(* CODESYS project Git_Repo
   Author: SESA110233
   DefaultNamespace: CrankModuleExample
   Title: Template_GitHub_ESME22
   Version: 0.0.0.0

Project tree, tasks and I/O mapping:
  LMC_PacDrive : PacDrive LMC 300/400/402/600/802/902C, Schneider Electric, order no. LMC Pro and Pro2, version 1.76.4.3
    application Application
      libraries: PD_GlobalDiagnostics, 1.6.0.0 (Schneider Electric); PD_PacDriveLib, 1.10.3.0 (Schneider Electric); PD_Template, 1.8.0.0 (Schneider Electric); PD_AxisModule, 1.7.1.0 (Schneider Electric); CrankModule, 1.4.1.0 (Schneider Electric); ApplicationLogger, 1.1.7.0 (Schneider Electric); IecRtsServices, 1.0.5.0 (Schneider Electric)
      task TASK_SR_Diagnostics (cyclic, interval T#100ms, priority 31, watchdog T#100ms x 2) calls SR_Diagnostics
      task TASK_SR_Logging (cyclic, interval T#10ms, priority 13, watchdog T#10ms x 2) calls SR_Logging
      task TASK_SR_MainMachine (cyclic, interval T#10ms, priority 8, watchdog t#10ms x 10) calls SR_HWCopyIO, SR_MainMachine
      task TASK_SR_VisControl (cyclic, interval T#50ms, priority 14, watchdog T#50ms x 2) calls SR_VisControl
      function CheckBounds [ST]
      function CheckDivDInt [ST]
      function CheckDivLInt [ST]
      function CheckDivLReal [ST]
      function CheckDivReal [ST]
      function CheckLRangeSigned [ST]
      function CheckLRangeUnsigned [ST]
      function CheckPointer [ST]
      function CheckRangeSigned [ST]
      function CheckRangeUnsigned [ST]
      CrankModuleExample/
        EquipmentModules/
          program SR_AlphaModule [SFC]: ExceptionControl_Action, Init_CmdTables, Init_Exceptions, Init_Master, Init_Reactions, Init_SubModules, InitModule_Action, Input_Action, Logger_Action, ModuleFaults, Output_Active, Start_Action, SubModules_Action, UpdateStructs
          program SR_BravoModule [SFC]: ExceptionControl_Action, Init_CmdTables, Init_Exceptions, Init_Reactions, Init_Slave1, Init_Slave2, Init_SubModules, InitModule_Action, Input_Action, Logger_Action, ModuleFaults, Output_Active, Start_Action, SubModules_Action, UpdateStructs
          program SR_CharlyModule [SFC]: ExceptionControl_Action, Init_CmdTables, Init_CrankModule, Init_Exceptions, Init_Nocke1, Init_Reactions, Init_Slave3, Init_Slave4, Init_SubModules, InitModule_Action, Input_Action, Logger_Action, Logic_Action, ModuleFaults, Output_Active, Start_Action, SubModules_Action, UpdateStructs
          program SR_NodeWithoutMotionModule [SFC]: ExceptionControl_Action, Init_CmdTables, Init_Exceptions, Init_Reactions, Init_SubModules, InitModule_Action, Input_Action, Logger_Action, ModuleFaults, Output_Active, Start_Action, SubModules_Action, UpdateStructs
        Examples/
          ExampleCmds/
            data type ET_Cmd
          ExampleModulesExtItf/
            function block FB_AxisModuleExtItf [ST]
            function block FB_ExampleLeafModuleExtItf [ST]
            function block FB_ExampleNodeFbModuleExtItf [ST]
            program SR_CharlyModuleExtItf [ST]
          ExampleNodeAsFB/
            function block FB_ExampleNodeFbModule [SFC]: ExceptionControl_Action, Init_CmdTables, Init_Exceptions, Init_Reactions, Init_Slave1, Init_Slave2, Init_SubModules, InitModule_Action, Input_Action, Logger_Action, ModuleFaults, Output_Active, Start_Action, SubModules_Action, UpdateStructs
            data type ST_ExampleNodeAsFbInterface
        GlobalVariables/
          global variables Diagnostics
          global variables ExceptionHandling
          global variables HardwareInOuts
          global variables InputVariablesEpas
          global variables InputVariablesExt
          global variables IntelligentLineShaft
          global variables Logging
          global variables RestoreAxisPosition
        ProjectDiagnostics/
          data type ET_DiagExt
          data type ET_DiagExtUser
          function FC_EtDiagExtToString [ST]
          function FC_EtDiagExtUserToString [ST]
        TaskCalls/
          program SR_Diagnostics [FBD]: SetDiagnosticsWarning
          program SR_HWCopyIO [FBD]
          program SR_Logging [FBD]
          program SR_MainMachine [SFC]: _aStart_active, AutoStep_Action, AutoStep_Entry, AutoStop_Action, AutoStop_Entry, BrakeReleaseStep_Action, BrakeReleaseStep_Entry, ExceptionControl_Action, Init_Alpha, Init_Bravo, Init_Charly, Init_CmdTables, Init_Exceptions, Init_NodeWithoutMotion, Init_Reactions, Init_SubModules, InitModule_Action, Input_Action, JogMachineStep_Action, JogMachineStep_Entry, Logger_Action, Logic_active, MainSystemFaults, MainUserFaults, ManualStep_Action, ManualStep_Entry, ModeSelect_Action, Output_Action, PrepStep_Action, PrepStep_Entry, PrepStop_Action, PrepStop_Entry, StopBrake_Action, StopBrake_Entry, StopJog_Action, StopJog_Entry, StopMan_Action, StopMan_Entry, SubModules_Action, UpdateStructs
          program SR_VisControl [ST]: CallTestErrors, CrankModuleVis, CurrentModuleCmdTable, DetectOpModeChange, ExceptionVis, InitTestExceptions, LoggerVis, MainPageCmdTable, ModuleNavigationIn, ModuleNavigationOut, ModuleReaction, ModuleVisController, OpModeControl, SearchCurrentModule, SetCurrentModule
        Tools/
          function FC_IsDriveVirtual [ST]
          function FC_SetDeadTimeCompensation [ST]
        Visualization/
          CrankModule/
            visualisation VIS_CrankModule
          visualisation VIS_Main
      function block FB_ExampleTableDiagSource [ST]: CancelWriting, ExceptionDuringWriting, SetDiagOutputs
      function block FB_ExampleTreeDiagSource [ST]: CancelWriting, ExceptionDuringWriting, SetDiagOutputs
      data type ET_DiagExtExampleLeafModule
      data type ET_ExampleLeafModuleCmd
      data type ET_ExampleLeafModuleState
      data type ET_ExceptionSource
      data type ET_ModuleType
      function block FB_ExampleLeafModule [SFC]: Auto_Action, Auto_Entry, CancelException, CheckCmd, CmdControl_Action, DiagQuit, DisableAllJobs, ExceptionHandler_Action, Homing_Action, Homing_Entry, InactiveCmdExecution, Init_Action, InitHoming_Action, InitHoming_Entry, Input_Action, Logger_Action, NoOp_Entry, Output_Active, RefuseCommand, ReportException, SetInterfaces, SetOutputs, SignalSuccessfulExecution, SignalUnSuccessfulExecution
      function block FB_ExampleLeafModuleController [ST]
      function block FB_ExampleLeafModuleVisController [ST]
      function FC_EtDiagExtExampleLeafModuleToString [ST]
      function FC_EtExampleLeafModuleCmdToString [ST]
      function FC_EtExampleLeafModuleStateToString [ST]
      function FC_UpdateExampleLeafModuleAddInterfaceStruct [ST]
      data type ST_ExampleLeafModuleInterface
      visualisation FR_ButtonAssignId
      visualisation FR_ExampleLeafModule
      visualisation FR_ExampleLeafModuleSelect
      visualisation VIS_ExampleLeafModule
      visualisation FR_ControlModuleTypes
      visualisation FR_NavigationButtons
      visualisation FR_OtherModuleTypes
      visualisation VIS_AxisModule
      visualisation VIS_ControlModule
      visualisation VIS_ExceptionDetails
      visualisation VIS_ExceptionList
      visualisation VIS_LogDataList
      visualisation VIS_LogDataListExt
      visualisation VIS_ModuleDetails
      visualisation VIS_ModuleExceptions
      visualisation VIS_Modules
      visualisation VIS_VisNavigation
    Device Addressing
    Message Logger
    AI_0 : Analog Input, Schneider Electric, version 1.76.4.3
    AI_1 : Analog Input, Schneider Electric, version 1.76.4.3
    AQ_0 : Analog Output, Schneider Electric, version 1.76.4.3
    AQ_1 : Analog Output, Schneider Electric, version 1.76.4.3
    DIG_DigitalIn : Digital Inputs, Schneider Electric, version 1.76.4.3
      DI_0 : Input, Schneider Electric, version 1.76.4.3
      DI_10 : Input, Schneider Electric, version 1.76.4.3
      DI_11 : Input, Schneider Electric, version 1.76.4.3
      DI_12 : Input, Schneider Electric, version 1.76.4.3
      DI_13 : Input, Schneider Electric, version 1.76.4.3
      DI_14 : Input, Schneider Electric, version 1.76.4.3
      DI_15 : Input, Schneider Electric, version 1.76.4.3
      DI_16 : Input, Schneider Electric, version 1.76.4.3
      DI_17 : Input, Schneider Electric, version 1.76.4.3
      DI_18 : Input, Schneider Electric, version 1.76.4.3
      DI_19 : Input, Schneider Electric, version 1.76.4.3
      DI_1 : Input, Schneider Electric, version 1.76.4.3
      DI_2 : Input, Schneider Electric, version 1.76.4.3
      DI_3 : Input, Schneider Electric, version 1.76.4.3
      DI_4 : Input, Schneider Electric, version 1.76.4.3
      DI_5 : Input, Schneider Electric, version 1.76.4.3
      DI_6 : Input, Schneider Electric, version 1.76.4.3
      DI_7 : Input, Schneider Electric, version 1.76.4.3
      DI_8 : Input, Schneider Electric, version 1.76.4.3
      DI_9 : Input, Schneider Electric, version 1.76.4.3
      FI_0 : Fast Input, Schneider Electric, version 1.76.4.3
      FI_1 : Fast Input, Schneider Electric, version 1.76.4.3
      FI_2 : Fast Input, Schneider Electric, version 1.76.4.3
      FI_3 : Fast Input, Schneider Electric, version 1.76.4.3
    DQG_DigitalOut : Digital Outputs, Schneider Electric, version 1.76.4.3
        settings: OpenloadDiagMsk = 0
      DQ_0 : Output, Schneider Electric, version 1.76.4.3
      DQ_10 : Output, Schneider Electric, version 1.76.4.3
      DQ_11 : Output, Schneider Electric, version 1.76.4.3
      DQ_12 : Output, Schneider Electric, version 1.76.4.3
      DQ_13 : Output, Schneider Electric, version 1.76.4.3
      DQ_14 : Output, Schneider Electric, version 1.76.4.3
      DQ_15 : Output, Schneider Electric, version 1.76.4.3
      DQ_1 : Output, Schneider Electric, version 1.76.4.3
      DQ_2 : Output, Schneider Electric, version 1.76.4.3
      DQ_3 : Output, Schneider Electric, version 1.76.4.3
      DQ_4 : Output, Schneider Electric, version 1.76.4.3
      DQ_5 : Output, Schneider Electric, version 1.76.4.3
      DQ_6 : Output, Schneider Electric, version 1.76.4.3
      DQ_7 : Output, Schneider Electric, version 1.76.4.3
      DQ_8 : Output, Schneider Electric, version 1.76.4.3
      DQ_9 : Output, Schneider Electric, version 1.76.4.3
    LE_EncCrank : Log. Encoder, Schneider Electric, version 1.76.4.3
    LE_EncSlide : Log. Encoder, Schneider Electric, version 1.76.4.3
    LE_Master : Log. Encoder, Schneider Electric, version 1.76.4.3
    LE_Slave1 : Log. Encoder, Schneider Electric, version 1.76.4.3
    LE_Slave2 : Log. Encoder, Schneider Electric, version 1.76.4.3
    LE_Slave3 : Log. Encoder, Schneider Electric, version 1.76.4.3
    LE_Slave4 : Log. Encoder, Schneider Electric, version 1.76.4.3
    Sercos_Master : Sercos Master, Schneider Electric, version 1.76.4.3
      DRV_CrankDrive : Lexium LXM62 Drive, Schneider Electric, order no. LXM62DU60, LXM62DD15, LXM62DD27, LXM62DD45, LXM62DC13, version 1.76.4.3
      DRV_Master : Lexium LXM62 Drive, Schneider Electric, order no. LXM62DU60, LXM62DD15, LXM62DD27, LXM62DD45, LXM62DC13, version 1.76.4.3
      DRV_Slave1 : Lexium LXM62 Drive, Schneider Electric, order no. LXM62DU60, LXM62DD15, LXM62DD27, LXM62DD45, LXM62DC13, version 1.76.4.3
      DRV_Slave2 : Lexium LXM62 Drive, Schneider Electric, order no. LXM62DU60, LXM62DD15, LXM62DD27, LXM62DD45, LXM62DC13, version 1.76.4.3
      DRV_Slave3 : Lexium LXM62 Drive, Schneider Electric, order no. LXM62DU60, LXM62DD15, LXM62DD27, LXM62DD45, LXM62DC13, version 1.76.4.3
      DRV_Slave4 : Lexium LXM62 Drive, Schneider Electric, order no. LXM62DU60, LXM62DD15, LXM62DD27, LXM62DD45, LXM62DC13, version 1.76.4.3
      DRV_SlideDrive : Lexium LXM62 Drive, Schneider Electric, order no. LXM62DU60, LXM62DD15, LXM62DD27, LXM62DD45, LXM62DC13, version 1.76.4.3
      PSM_PowerSupply : Lexium LXM62 Power Supply, Schneider Electric, order no. LXM62PD84, LXM62PD20, version 1.76.4.3
    TPG_TPIn : Touch Probe Inputs, Schneider Electric, version 1.76.4.3
      TP_0 : Touch Probe Input, Schneider Electric, version 1.76.4.3
      TP_10 : Touch Probe Input, Schneider Electric, version 1.76.4.3
      TP_11 : Touch Probe Input, Schneider Electric, version 1.76.4.3
      TP_12 : Touch Probe Input, Schneider Electric, version 1.76.4.3
      TP_13 : Touch Probe Input, Schneider Electric, version 1.76.4.3
      TP_14 : Touch Probe Input, Schneider Electric, version 1.76.4.3
      TP_15 : Touch Probe Input, Schneider Electric, version 1.76.4.3
      TP_1 : Touch Probe Input, Schneider Electric, version 1.76.4.3
      TP_2 : Touch Probe Input, Schneider Electric, version 1.76.4.3
      TP_3 : Touch Probe Input, Schneider Electric, version 1.76.4.3
      TP_4 : Touch Probe Input, Schneider Electric, version 1.76.4.3
      TP_5 : Touch Probe Input, Schneider Electric, version 1.76.4.3
      TP_6 : Touch Probe Input, Schneider Electric, version 1.76.4.3
      TP_7 : Touch Probe Input, Schneider Electric, version 1.76.4.3
      TP_8 : Touch Probe Input, Schneider Electric, version 1.76.4.3
      TP_9 : Touch Probe Input, Schneider Electric, version 1.76.4.3
  00000000-0000-0000-0000-000000000000|M:\lib-jenkins-config\externalfiles\Disclaimer of Warranty.pdf
  Disclaimer of Warranty
  text list GlobalTextList
  function GetBooleanProperty [ST]
  function GetTextProperty2 [ST]
  function GetTextProperty [ST]
  function GetTitle [ST]
*)

// LMC_PacDrive/Application/CrankModuleExample/ProjectDiagnostics/ET_DiagExt
{attribute 'qualified_only'}
TYPE ET_DiagExt :
(
	(* Minimum value +0 *)
	Ok								:= 0,
	Disabled						:= 1,
	WaitUntilControllerFinishedBoot	:= 2,
	Initializing					:= 3,
	DeactivatingSubModules			:= 4,
	ExecuteStep						:= 5,
	WaitAtNegativeStep				:= 6,
	WaitCmdsDone					:= 7,
	WaitForCmd						:= 8,
	SubModuleInException			:= 9,
	ModuleControllerException		:= 10,
	UnknownStateModuleController	:= 11,
	
	SystemFatalException			:= 12,
	SystemException					:= 13,
	SystemWarning					:= 14,
	MainSystemEmergencyStop			:= 15,
	InvalidPointer					:= 16,	
	UpdateStructsException			:= 17,
	InitReactionsException			:= 18,
	InitSubModulesException			:= 19,
	DriveInvalid					:= 20,
	UnknownDiagExt					:= 21,
	
	Exception1FromVis				:= 22,
	Exception2FromVis				:= 23,
	Exception3FromVis				:= 24,
	Exception4FromVis				:= 25,
	Exception5FromVis				:= 26,
	
	DiagnosticsWarning					:= 27,
	WaitUntilDiagnosticsManagerReady	:= 28,
	WaitUntilDisabled					:= 29,
	WaitUntilDiagSourceRegistered		:= 30,
	WaitForCommunication				:= 31,
	DataSuccessfullyWritten				:= 32,
	WritingToFile						:= 33,
	FileIdInvalid						:= 34,
	CmdUnknown							:= 35,	
	UnexpectedFeedback					:= 36,
	UnknownDiagExtUser					:= 37
)UDINT;
END_TYPE

// LMC_PacDrive/Application/CrankModuleExample/ProjectDiagnostics/ET_DiagExtUser
{attribute 'qualified_only'}
TYPE ET_DiagExtUser :
(
(* Minimum value +0 *)
	Exception1FromEquipmentModule		:= 0,
	Exception2FromEquipmentModule		:= 1,
	
	Exception1FromMain					:= 2,
	Exception2FromMain					:= 3,
	Exception3FromMain					:= 4,
	Exception4FromMain					:= 5,
	Exception5FromMain					:= 6
)UDINT;
END_TYPE

// LMC_PacDrive/Application/CrankModuleExample/Examples/ExampleCmds/ET_Cmd
{attribute 'qualified_only'}
TYPE ET_Cmd :
(	NoCmd				:= 0,

	(* TPL.Gc_udiUserCmdOffset : UDINT := 25000; // >= 25000: user defined Commands *)
	DriveEnableOn		:= 25999,
	DriveEnableOff		:= 25998,
	Init				:= 25997,
	Prepare				:= 25996,
	Production			:= 25995,
	Auto				:= 25994,
	BrakeRelease		:= 25993,
	Abort				:= 25992,
	Standby				:= 25991,
	Manual				:= 25990,
	Jogging				:= 25989,
	Hold				:= 25988,
	Stop				:= 25987,
	Start				:= 25986,
	HoldJM				:= 25985
);
END_TYPE

// LMC_PacDrive/Application/ET_DiagExtExampleLeafModule
{attribute 'qualified_only'}
TYPE ET_DiagExtExampleLeafModule :
(
(* Minimum value +0 *)
	Ok										:= 0,
	Disabled								:= 1,
	Initializing							:= 2,
	NoOp									:= 3,
	HomingWaitForStart						:= 4,
	HomingExecuting							:= 5,
	HomingDone								:= 6,
	AutoWaitForStart						:= 7,
	AutoRunning								:= 8,
	Working									:= 9,

	UnknownDiagExtExampleLeafModule			:= 10,
	SubModuleAddInterfacesInvalidPointer	:= 11,
	SubModuleConstantRange					:= 12,
	MissingExtInit							:= 13,
	ReactionOffsetRange						:= 14,
	DriveInvalid							:= 15,
	
	CmdUnknown								:= 16,
	CmdImpossibleOverwrite					:= 17,
	CmdImpossibleState						:= 18,
	CmdImpossibleReaction					:= 19,
	
	AsyncStop								:= 20,
	SyncStopEL								:= 21,
	SyncStopEH								:= 22,
	StopEndOfCycle							:= 23,
	
	DriveFatalException						:= 24,
	DriveException							:= 25,
	DriveWarning							:= 26,
	
	UnknownState							:= 27,
	UnknownCmd								:= 28,
	RandomException							:= 29,
	
	CurrentStandardItfInvalidPointer		:= 30,
	CurrentAddItfInvalidPointer				:= 31
)UDINT;
END_TYPE

// LMC_PacDrive/Application/ET_ExampleLeafModuleCmd
{attribute 'qualified_only'}
TYPE ET_ExampleLeafModuleCmd :
(
	(* TPL.Gc_udiUserCmdOffset : UDINT := 25000; // >= 25000: user defined Commands *)
	Homing				:= 30000,
	Auto				:= 30001,
	Start				:= 30002,
	Stop				:= 30003,
	Hold				:= 30004
	
)DINT; //UDINT;
END_TYPE

// LMC_PacDrive/Application/ET_ExampleLeafModuleState
{attribute 'qualified_only'}
TYPE ET_ExampleLeafModuleState :
(
	NoOp				:= 0,
	Disabled			:= 1,
	Initializing		:= 2,
	HomingWaitForStart	:= 3,
	HomingExecuting		:= 4,
	HomingDone			:= 5,
	AutoWaitForStart	:= 6,
	AutoRunning			:= 7
)UDINT;
END_TYPE

// LMC_PacDrive/Application/ET_ExceptionSource
{attribute 'qualified_only'}
TYPE ET_ExceptionSource :
(
	(* 0 - 9999 = reserved area *)
	
	(* Sources > 9999 = free Area *)
	ExampleLeafModule	:= 15000
)UDINT;
END_TYPE

// LMC_PacDrive/Application/ET_ModuleType
{attribute 'qualified_only'}
TYPE ET_ModuleType :
(
	(* 0 - 9999 = reserved area *)
	(* IDs >9999 = free Area *)
	ExampleLeafModule := 15000 (* Definition of the dwModuleType for the module *)
)UDINT;
END_TYPE

// LMC_PacDrive/Application/ST_ExampleLeafModuleInterface
TYPE ST_ExampleLeafModuleInterface :
STRUCT
	i_ifDrive						: SystemConfigurationItf.IF_Drive;
	i_lrPosMin						: LREAL;
	i_lrPosMax						: LREAL;
	i_xInitHoming					: BOOL;
	i_xEnableRandomExceptionTrigger	: BOOL;
	
	q_xValue						: BOOL := FALSE;
	q_etState						: ET_ExampleLeafModuleState := ET_ExampleLeafModuleState.Disabled;
END_STRUCT
END_TYPE

// LMC_PacDrive/Application/CrankModuleExample/Examples/ExampleNodeAsFB/ST_ExampleNodeAsFbInterface
TYPE ST_ExampleNodeAsFbInterface :
STRUCT
	i_ifSlave1				: SystemConfigurationItf.IF_Drive;
	i_lencEncoder1			: SystemConfiguration.L_ENC;
	i_ifHomingTouchProbe1	: SystemConfigurationItf.IF_TouchProbe;
	i_pstRestorePosRetain1	: POINTER TO PDL.ST_AxisRestorePosition;
	
	i_ifSlave2				: SystemConfigurationItf.IF_Drive;
	i_lencEncoder2			: SystemConfiguration.L_ENC;
	i_ifHomingTouchProbe2	: SystemConfigurationItf.IF_TouchProbe;
	i_pstRestorePosRetain2	: POINTER TO PDL.ST_AxisRestorePosition;
END_STRUCT
END_TYPE

// LMC_PacDrive/Application/CrankModuleExample/GlobalVariables/Diagnostics
VAR_GLOBAL
	G_stDiagnosticsToApplicationMarkerarea AT %MB0 : TPL.ST_DiagnosticsToApplicationMarkerArea;
END_VAR

// LMC_PacDrive/Application/CrankModuleExample/GlobalVariables/ExceptionHandling
VAR_GLOBAL
	G_stExceptionList		: TPL.ST_ExceptionList;
END_VAR

// LMC_PacDrive/Application/CrankModuleExample/GlobalVariables/HardwareInOuts
VAR_GLOBAL
	G_xMainsContactorOut 		(*-AT %QX0.0-*)	: BOOL;

	G_xEmergencyIn  			(*-AT %IX0.0-*)	: BOOL;
	G_xMainsContactorIn 		(*-AT %IX0.1-*)	: BOOL;
END_VAR

// LMC_PacDrive/Application/CrankModuleExample/GlobalVariables/InputVariablesEpas
VAR_GLOBAL
	G_xStartEpas				: BOOL;
	G_xStopEpas					: BOOL;
	G_xPrepareEpas				: BOOL;
	G_xAutoEpas					: BOOL;
	G_xHoldEpas					: BOOL;
	G_xAbortEpas				: BOOL;
	G_xProductsOkEpas			: BOOL;
	G_xPowerOnEpas				: BOOL;
	G_xPowerOffEpas				: BOOL;
	G_xManualEpas				: BOOL;
	G_xJogMachineEpas			: BOOL;
	G_xDiagQuitEpas				: BOOL;
	G_xEmergencyEpas			: BOOL := TRUE;
	G_xJogForwEpas				: BOOL;
	G_xJogBackEpas				: BOOL;
	G_xBrakeReleaseEpas			: BOOL;
	
	G_udiManualModuleSelect		: UDINT;

	G_xDoEnableVis				: BOOL;
	
	G_xDoEnableCrankVis			: BOOL; // created for Crank execution.

	G_xDoPrepare 				: BOOL;
	G_xDoAuto	 				: BOOL;
	G_xDoManual 				: BOOL;
	G_xDoJogMachine 			: BOOL;
	G_xDoBrakeRelease			: BOOL;

	G_xPrepareActive 			: BOOL;
	G_xAutoActive	 			: BOOL;
	G_xManualActive 			: BOOL;
	G_xJogMachineActive 		: BOOL;
	G_xBrakeReleaseActive		: BOOL;
END_VAR

// LMC_PacDrive/Application/CrankModuleExample/GlobalVariables/InputVariablesExt
VAR_GLOBAL
	G_xStartExt			: BOOL;
	G_xStopExt			: BOOL;
	G_xPrepareExt		: BOOL;
	G_xAutoExt			: BOOL;
	G_xHoldExt			: BOOL;
	G_xAbortExt			: BOOL;
	G_xProductsOkExt	: BOOL;
	G_xPowerOnExt		: BOOL;
	G_xPowerOffExt		: BOOL;
	G_xManualExt		: BOOL;
	G_xJogMachineExt	: BOOL;
	G_xDiagQuitExt		: BOOL;
	G_xJogForwExt		: BOOL;
	G_xJogBackExt		: BOOL;
	G_xBrakeReleaseExt	: BOOL;
END_VAR

// LMC_PacDrive/Application/CrankModuleExample/GlobalVariables/IntelligentLineShaft
VAR_GLOBAL
	G_stIlsData : PDL.ST_IlsData;
END_VAR

// LMC_PacDrive/Application/CrankModuleExample/GlobalVariables/Logging
VAR_GLOBAL
	G_stLogDataList			: TPL.ST_LogDataList;			(* Global log data list *)
	G_stLogDataListAscii	: TPL.ST_LogDataListAscii;		(* Temp.list for save in XML format *)
	G_stLoggerInterface		: TPL.ST_LoggerInterface;		(* Interface between logger and main machine *)
END_VAR

// LMC_PacDrive/Application/CrankModuleExample/GlobalVariables/RestoreAxisPosition
VAR_GLOBAL PERSISTENT RETAIN
	Grp_stRestorePositionAxis1		: PDL.ST_AxisRestorePosition;
	Grp_stRestorePositionAxis2		: PDL.ST_AxisRestorePosition;
	Grp_stRestorePositionAxis3		: PDL.ST_AxisRestorePosition;
	Grp_stRestorePositionAxis4		: PDL.ST_AxisRestorePosition;
	Grp_stRestorePositionAxis5		: PDL.ST_AxisRestorePosition;
	Grp_stRestorePositionAxis6		: PDL.ST_AxisRestorePosition;
	Grp_stRestorePositionAxis7		: PDL.ST_AxisRestorePosition;
	Grp_stRestorePositionAxis8		: PDL.ST_AxisRestorePosition;
	Grp_stRestorePositionAxisCrank	: PDL.ST_AxisRestorePosition;
END_VAR

// LMC_PacDrive/Application/CrankModuleExample/TaskCalls/SR_Diagnostics
PROGRAM SR_Diagnostics
VAR
	fbDiagnosticsManager : TPL.FB_DiagnosticsManager;
	stComStructure 		 : TPL.ST_DiagnosticsManagerToDiagSource;
	
	stWarning 		: TPL.ST_Exception;
	etLastDiagExt	: TPL.ET_DiagExt := TPL.ET_DiagExt.Ok;

	(* Add the instances of your sources for diag data here *)
	fbTemplateStaticStructureDiagSource	: TPL.FB_TemplateStaticStructureDiagSource;
	fbExceptionListDiagSource			: TPL.FB_ExceptionListDiagSource;
	fbExceptionDelayListDiagSource		: TPL.FB_ExceptionDelayListDiagSource;
	fbLogDataListDiagSource				: TPL.FB_LogDataListDiagSource;	
	fbAxisModuleDiagSource				: AXM.FB_AxisModuleDiagSource;
	xPrintCamData						: BOOL := TRUE;
	fbCrankModuleDiagSource				: CRKM.FB_CrankModuleDiagSource;

	(* example diag sources *)
	fbExampleTableDiagSource			: FB_ExampleTableDiagSource;
	fbExampleTreeDiagSource				: FB_ExampleTreeDiagSource;
END_VAR

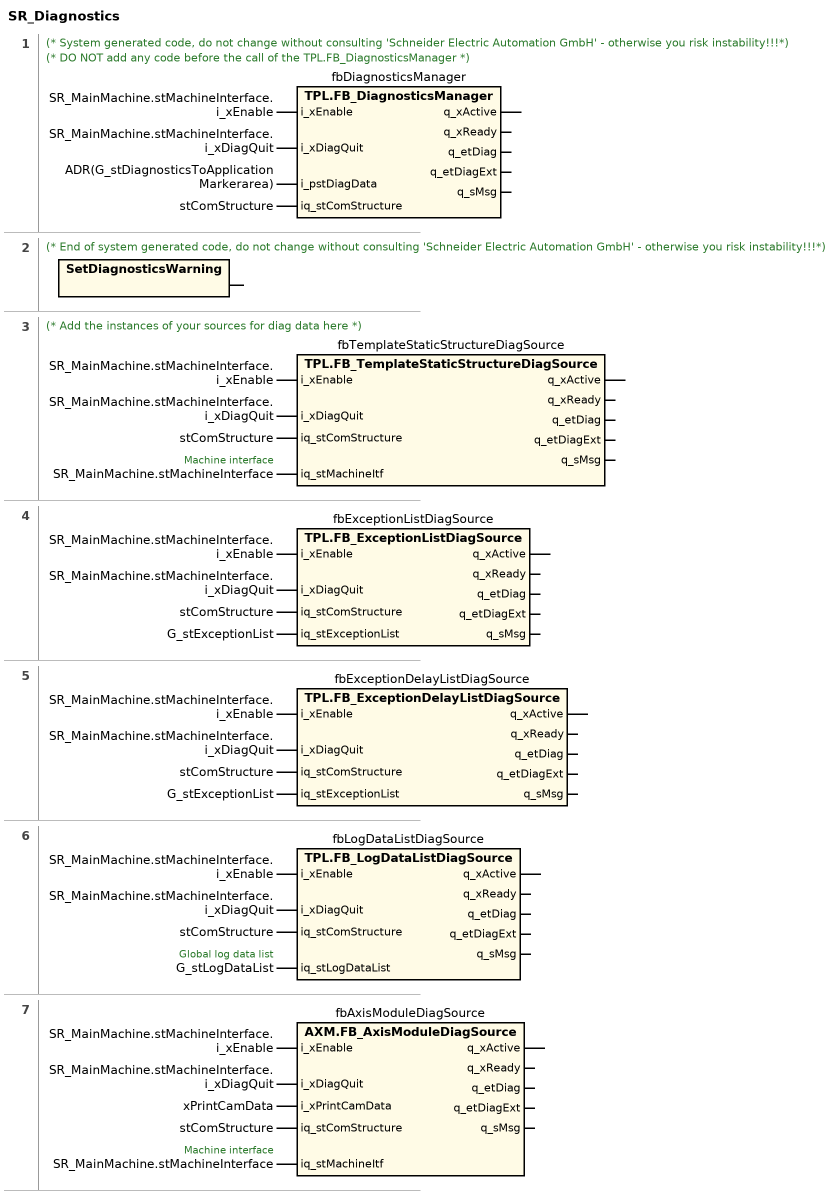
// NETWORK 1
// (* System generated code, do not change without consulting 'Schneider Electric Automation GmbH' - otherwise you risk instability!!!*)
// (* DO NOT add any code before the call of the TPL.FB_DiagnosticsManager *)
fbDiagnosticsManager(
    i_xEnable := SR_MainMachine.stMachineInterface.i_xEnable,
    i_xDiagQuit := SR_MainMachine.stMachineInterface.i_xDiagQuit,
    i_pstDiagData := ADR(G_stDiagnosticsToApplicationMarkerarea),
    iq_stComStructure := stComStructure); // TPL.FB_DiagnosticsManager

// NETWORK 2
// (* End of system generated code, do not change without consulting 'Schneider Electric Automation GmbH' - otherwise you risk instability!!!*)
SetDiagnosticsWarning();

// NETWORK 3
// (* Add the instances of your sources for diag data here *)
//   fbTemplateStaticStructureDiagSource: Add the instances of your sources for diag data here
//   SR_MainMachine.stMachineInterface: Machine interface
fbTemplateStaticStructureDiagSource(
    i_xEnable := SR_MainMachine.stMachineInterface.i_xEnable,
    i_xDiagQuit := SR_MainMachine.stMachineInterface.i_xDiagQuit,
    iq_stComStructure := stComStructure,
    iq_stMachineItf := SR_MainMachine.stMachineInterface); // TPL.FB_TemplateStaticStructureDiagSource

// NETWORK 4
fbExceptionListDiagSource(
    i_xEnable := SR_MainMachine.stMachineInterface.i_xEnable,
    i_xDiagQuit := SR_MainMachine.stMachineInterface.i_xDiagQuit,
    iq_stComStructure := stComStructure,
    iq_stExceptionList := G_stExceptionList); // TPL.FB_ExceptionListDiagSource

// NETWORK 5
fbExceptionDelayListDiagSource(
    i_xEnable := SR_MainMachine.stMachineInterface.i_xEnable,
    i_xDiagQuit := SR_MainMachine.stMachineInterface.i_xDiagQuit,
    iq_stComStructure := stComStructure,
    iq_stExceptionList := G_stExceptionList); // TPL.FB_ExceptionDelayListDiagSource

// NETWORK 6
//   G_stLogDataList: Global log data list
fbLogDataListDiagSource(
    i_xEnable := SR_MainMachine.stMachineInterface.i_xEnable,
    i_xDiagQuit := SR_MainMachine.stMachineInterface.i_xDiagQuit,
    iq_stComStructure := stComStructure,
    iq_stLogDataList := G_stLogDataList); // TPL.FB_LogDataListDiagSource

// NETWORK 7
//   SR_MainMachine.stMachineInterface: Machine interface
fbAxisModuleDiagSource(
    i_xEnable := SR_MainMachine.stMachineInterface.i_xEnable,
    i_xDiagQuit := SR_MainMachine.stMachineInterface.i_xDiagQuit,
    i_xPrintCamData := xPrintCamData,
    iq_stComStructure := stComStructure,
    iq_stMachineItf := SR_MainMachine.stMachineInterface); // AXM.FB_AxisModuleDiagSource

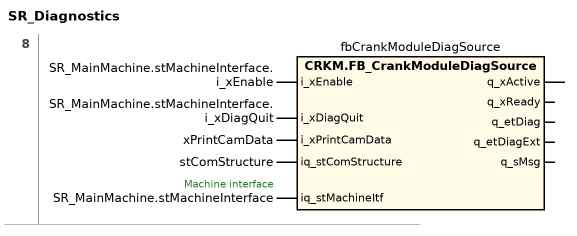
// NETWORK 8
//   SR_MainMachine.stMachineInterface: Machine interface
fbCrankModuleDiagSource(
    i_xEnable := SR_MainMachine.stMachineInterface.i_xEnable,
    i_xDiagQuit := SR_MainMachine.stMachineInterface.i_xDiagQuit,
    i_xPrintCamData := xPrintCamData,
    iq_stComStructure := stComStructure,
    iq_stMachineItf := SR_MainMachine.stMachineInterface); // CRKM.FB_CrankModuleDiagSource

ACTION SetDiagnosticsWarning:
(* System generated code, do not change without consulting 'Schneider Electric Automation GmbH' - otherwise you risk instability!!!*)
						
(* Signal exception during diagnostics, but as diagnostics should not influence the machine, create only a warning *)
IF(fbDiagnosticsManager.q_etDiag <> GD.ET_Diag.Ok AND fbDiagnosticsManager.q_etDiagExt <> etLastDiagExt) THEN
	
	stWarning.etDiag		:= GD.ET_Diag.DiagActive;
	stWarning.udiDiagExt	:= ET_DiagExt.DiagnosticsWarning;
	stWarning.sDiagExt		:= FC_EtDiagExtToString(ET_DiagExt.DiagnosticsWarning);
	stWarning.udiModuleId	:= SR_MainMachine.c_udiMainModuleId;
	stWarning.sMsg			:= CONCAT(CONCAT('SR_Diagnostics: ', GD.FC_EtDiagToString(fbDiagnosticsManager.q_etDiag)), CONCAT(' ; ', TPL.FC_EtDiagExtToString(fbDiagnosticsManager.q_etDiagExt)));
	stWarning.sModuleName	:= SR_MainMachine.stMachineInterface.i_sModuleName;
	stWarning.etSource		:= TPL.ET_ExceptionSource.Logger;
	
	TPL.FC_SetException(	i_xExceptionActive	:= TRUE,
							iq_stException		:= stWarning,
							iq_stExceptionList	:= G_stExceptionList,
							iq_stLogDataList	:= G_stLogDataList);
END_IF

etLastDiagExt := fbDiagnosticsManager.q_etDiagExt;
(* End of system generated code, do not change without consulting 'Schneider Electric Automation GmbH' - otherwise you risk instability!!!*)
END_ACTION

END_PROGRAM

// LMC_PacDrive/Application/CrankModuleExample/TaskCalls/SR_MainMachine
PROGRAM  SR_MainMachine

VAR CONSTANT
	c_udiNumberOfGroups			: UDINT := 3;		(* Maximum number of groups *)
	c_udiNumberOfGroupMembers	: UDINT := 3;		(* Maximum number of members per group *)

	c_udiNumberOfCmdTables		: UDINT := 10;		(* Must be the exact number of used CMDTables! *)
	c_udiNumberOfCmdSteps		: UDINT := 16;		(* Make sure that the number of command steps that each table
													   contains does not exceed the c_udiNumberOfCmdSteps variable.*)

(* Definition group of modules *)
	c_udiMasterGroup			: UDINT := 2001;	(* Name of module group  1 *)
	c_udiSlaveGroup				: UDINT := 2002;	(* Name of module group  2 *)

(* ModuleId of MainMachine *)
	c_udiMainModuleId			: UDINT := 1;		(* ModuleId *)

(* System generated code, could be modified for your application *)
	c_udiNumberOfSubModules		: UDINT := 4;		(* Number of SubModules *)
	c_udiAlpha					: UDINT := 1;		(* Name & number of Module 1 *)
	c_udiBravo					: UDINT := 2;		(* Name & number of Module 2 *)
	c_udiCharly					: UDINT := 3;		(* Name & number of Module 3 *)
	c_udiNodeWithoutMotion		: UDINT := 4;		(* Name & number of Module 4 *)

	c_dwModuleType				: DWORD := TPL.ET_ModuleType.MachineModule;
	c_sModuleTypeName			: STRING[14] := 'MainMachine';
	c_udiModuleVersion			: UDINT := 1;
(* End of system generated code, could be modified for your application *)
END_VAR

VAR (* User specific variables *)

END_VAR

VAR
	xInitSuccessful : BOOL := TRUE;
		
(*INPUT Variables*)
	xInputErrorQuit				: BOOL;
	xInputStart					: BOOL;
	xInputStop					: BOOL;
	xInputPrepare				: BOOL;
	xInputAuto					: BOOL;
	xInputManual				: BOOL;
	xInputJogMachine			: BOOL;
	xInputHold					: BOOL;
	xInputAbort					: BOOL;
	xInputProductsOk			: BOOL;
	xInputPowerOn				: BOOL;
	xInputPowerOff				: BOOL;
	xInputBrakeRelease			: BOOL;
	xInputEmergency				: BOOL := TRUE;

(* OUTPUT Variables *)
	xOutputPrepareActive		: BOOL;
	xOutputAutoActive			: BOOL;
	xOutputHoldActive			: BOOL;
	xOutputServiceActive		: BOOL;
	xOutputManualActive			: BOOL;
	xOutputJogMachineActive		: BOOL;

(* User Exceptions declaration *)
	stSystemException1				: TPL.ST_Exception;
	stSystemException2				: TPL.ST_Exception;
	stSystemException3				: TPL.ST_Exception;
	
	stEmergencyStopException		: TPL.ST_Exception;
	stContactorControlException		: TPL.ST_Exception;
	
	stUpdateStructsException		: TPL.ST_Exception;
	xUpdateStructsException			: BOOL;
	
	stInitReactionsException		: TPL.ST_Exception;
	xInitReactionsException			: BOOL;
	
	stInitSubModulesException		: TPL.ST_Exception;
	xInitSubModulesException		: BOOL;
	
	stUserException1				: TPL.ST_Exception;
	stUserException2				: TPL.ST_Exception;
	stUserException3				: TPL.ST_Exception;
	stUserException4				: TPL.ST_Exception;
	stUserException5				: TPL.ST_Exception;

	etSetExceptionDiag1			: GD.ET_Diag;
	etSetExceptionDiag2			: GD.ET_Diag;
	etSetExceptionDiag3			: GD.ET_Diag;
	etSetExceptionDiag4			: GD.ET_Diag;
	etSetExceptionDiag5			: GD.ET_Diag;
	
	etSetExceptionDiagExt1		: TPL.ET_DiagExt;
	etSetExceptionDiagExt2		: TPL.ET_DiagExt;
	etSetExceptionDiagExt3		: TPL.ET_DiagExt;
	etSetExceptionDiagExt4		: TPL.ET_DiagExt;
	etSetExceptionDiagExt5		: TPL.ET_DiagExt;
	
	etSetExceptionMsg1			: STRING[80];
	etSetExceptionMsg2			: STRING[80];
	etSetExceptionMsg3			: STRING[80];
	etSetExceptionMsg4			: STRING[80];
	etSetExceptionMsg5			: STRING[80];

(* OPM control Variables *)
	xActPrepare					: BOOL;
	xActAuto					: BOOL;
	xActManual					: BOOL;
	xActJogMachine				: BOOL;
	xActBrake					: BOOL;
	xCmdWasActive				: BOOL;

	xModeReady					: BOOL;
	xBrakeReady					: BOOL;
	xExitStop					: BOOL;

(* Main ModuleController *)
	fbModuleController				: TPL.FB_ModuleController;
	etDiagModuleController			: GD.ET_Diag;
	etDiagExtModuleController		: TPL.ET_DiagExt;
	sMsgModuleController			: STRING[80];
	xWaitForStartStep				: BOOL;

(* Standard related variables *)
	astSubModuleInterface		: ARRAY[1..c_udiNumberOfSubModules] OF TPL.ST_StandardModuleInterface;	(* Standard Module interface *)
	aaudiSubModuleGroups		: ARRAY[1..c_udiNumberOfGroups,1..c_udiNumberOfGroupMembers] OF UDINT;
	adwSubModuleAddInterfaces	: ARRAY[1..c_udiNumberOfSubModules] OF DWORD;
	
(* Machine interface *)
	stMachineInterface			: TPL.ST_StandardModuleInterface;
	stMachineMotionInterface	: TPL.ST_StandardMotionInterface;

(* Command table list *)
	astListofCMDTables			: ARRAY [1..c_udiNumberOfCmdTables] OF TPL.ST_CmdTable;   (* Cmd list of tables*)
	udiTableIndex				: UDINT;
	udiStepIndex				: UDINT;
	diStep						: DINT;
	
	astPrepareTable				: ARRAY [1..c_udiNumberOfCmdSteps] OF TPL.ST_Cmd; (* Relating  Cmd table *)
	astAutoTable				: ARRAY [1..c_udiNumberOfCmdSteps] OF TPL.ST_Cmd; (* Relating  Cmd table *)
	astManualTable				: ARRAY [1..c_udiNumberOfCmdSteps] OF TPL.ST_Cmd; (* Relating  Cmd table *)
	astHoldTable				: ARRAY [1..c_udiNumberOfCmdSteps] OF TPL.ST_Cmd; (* Relating  Cmd table *)
	astHoldJogMachineTable		: ARRAY [1..c_udiNumberOfCmdSteps] OF TPL.ST_Cmd; (* Relating  Cmd table *)
	astStartTable				: ARRAY [1..c_udiNumberOfCmdSteps] OF TPL.ST_Cmd; (* Relating  Cmd table *)
	astStopTable				: ARRAY [1..c_udiNumberOfCmdSteps] OF TPL.ST_Cmd; (* Relating  Cmd table *)
	astBrakeReleaseTable		: ARRAY [1..c_udiNumberOfCmdSteps] OF TPL.ST_Cmd; (* Relating  Cmd table *)
	astAbortTable				: ARRAY [1..c_udiNumberOfCmdSteps] OF TPL.ST_Cmd; (* Relating  Cmd table *)
	astJogMachineTable			: ARRAY [1..c_udiNumberOfCmdSteps] OF TPL.ST_Cmd; (* Relating  Cmd table *)

(* ExceptionHandling related variables *)
	fbExceptionHandler				: TPL.FB_ExceptionHandler;

	aetReactionTranslationMode		: ARRAY[1..c_udiNumberOfSubModules] OF TPL.ET_ReactionTranslationMode;
	aastReactionTranslationTable	: ARRAY[1..c_udiNumberOfSubModules,1..TPL.Gc_udiMaxNumberOfReactions] OF TPL.ST_Reaction;
	astReactionTranslationJobs		: ARRAY[1..c_udiNumberOfSubModules] OF TPL.ST_ReactionTranslationJobs;

	xCheckExceptionList				: BOOL := TRUE;
	xReactionActive					: BOOL;

	sDiagMsg						: STRING[120];
	xVirtualSystem					: BOOL;

(* Contactor Control related variables *)
	fbContactorControl			: TPL.FB_ContactorControl;
	xMainsOn					: BOOL := TRUE;
	xMainsWatch					: BOOL;
	timPowerOnDelay				: TIME := T#500MS;

	xContactorControlActive				: BOOL;
	xContactorControlReady				: BOOL;
	etContactorControlDiag				: GD.ET_Diag;		
	etContactorControlDiagExt			: TPL.ET_DiagExt;
	sContactorControlMsg				: STRING[80];
	xContactorControlPowerOnDelayOver	: BOOL;

(* Logging related variables*)
	fbLogger					: TPL.FB_Logger;

(* OnlineChange related variables *)
	fbDetectOnlineChange			: TPL.FB_DetectOnlineChange;
	xDetectOnlineChangeActive		: BOOL; 
	xDetectOnlineChangeReady		: BOOL; 
	etDetectOnlineChangeDiag		: GD.ET_Diag;
	etDetectOnlineChangeDiagExt		: TPL.ET_DiagExt; 
	sDetectOnlineChangeMsg			: STRING[80];

(* Exception  *)
	xTestUserException1				: BOOL;
	xTestUserException2				: BOOL;
	xTestUserException3				: BOOL;
	xTestUserException4				: BOOL;
	xTestUserException5				: BOOL;

	iTemp						: INT;
	diClassTemp					: DINT;

	fbControllerDiag			: TPL.FB_ControllerDiag;
	diObjectType				: DINT;								(* Diag: Object No. *)
	sTypeName					: STRING[10];						(* Diag: Object Name *)
	diObjectInstance			: DINT;								(* Diag: Instance No. *)
	sInstanceName				: STRING[40];						(* Diag: Instance Name *)
	diDiagCode					: DINT;								(* Diag: Class and Number *)
	diDiagClass					: DINT;								(* Diag: Class *)
	diDiagNum					: DINT;								(* Diag: Number *)
	sDiagText					: STRING[40];						(* Diag: Text *)
	xHWReset					: BOOL;								(* Diag: Hardware reset necessary *)
	
(* POU-Feedback related variables*)	
	etDiag			: GD.ET_Diag;
	etDiagExt		: ET_DiagExt;
	etDiagExtTPL	: TPL.ET_DiagExt;
	etDiagExtAXM	: AXM.ET_DiagExt;
	
(* GitHub *)
	xPaolo			: BOOL;
	
END_VAR
VAR // added by the converter: edge detectors and wires of the graphical bodies
    _w1 : BOOL;
END_VAR

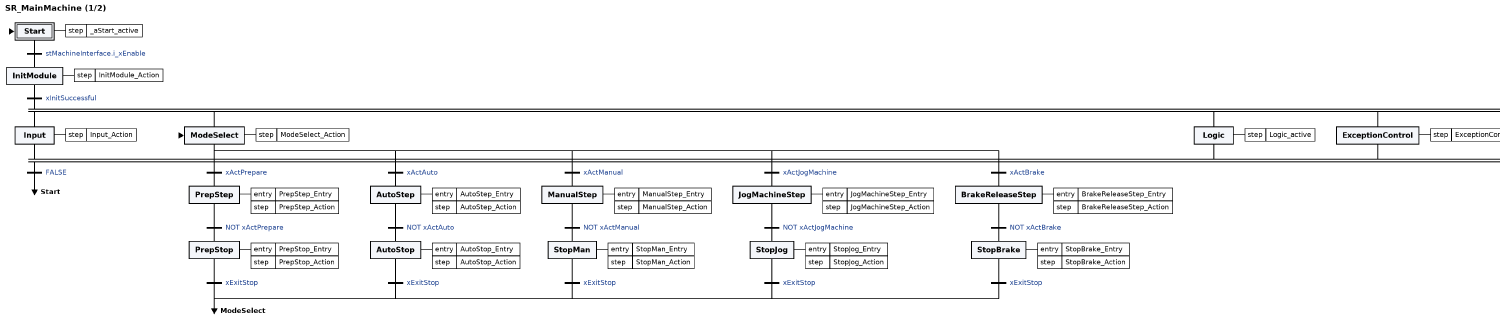
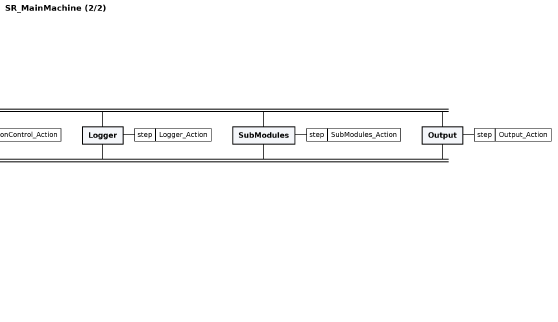
INITIAL_STEP Start:
    _aStart_active(N);  // step action
END_STEP
TRANSITION FROM Start TO InitModule
    := stMachineInterface.i_xEnable;
END_TRANSITION
STEP InitModule:
    InitModule_Action(N);  // step action
END_STEP
TRANSITION FROM InitModule TO (Input, ModeSelect, Logic, ExceptionControl, Logger, SubModules, Output)
    := xInitSuccessful;
END_TRANSITION
STEP Input:
    Input_Action(N);  // step action
END_STEP
STEP ModeSelect:
    ModeSelect_Action(N);  // step action
END_STEP
TRANSITION FROM ModeSelect TO PrepStep
    := xActPrepare;
END_TRANSITION
STEP PrepStep:
    PrepStep_Entry(P1);  // entry action
    PrepStep_Action(N);  // step action
END_STEP
TRANSITION FROM PrepStep TO PrepStop
    := NOT xActPrepare;
END_TRANSITION
STEP PrepStop:
    PrepStop_Entry(P1);  // entry action
    PrepStop_Action(N);  // step action
END_STEP
TRANSITION FROM PrepStop TO ModeSelect
    := xExitStop;
END_TRANSITION
TRANSITION FROM ModeSelect TO AutoStep
    := xActAuto;
END_TRANSITION
STEP AutoStep:
    AutoStep_Entry(P1);  // entry action
    AutoStep_Action(N);  // step action
END_STEP
TRANSITION FROM AutoStep TO AutoStop
    := NOT xActAuto;
END_TRANSITION
STEP AutoStop:
    AutoStop_Entry(P1);  // entry action
    AutoStop_Action(N);  // step action
END_STEP
TRANSITION FROM AutoStop TO ModeSelect
    := xExitStop;
END_TRANSITION
TRANSITION FROM ModeSelect TO ManualStep
    := xActManual;
END_TRANSITION
STEP ManualStep:
    ManualStep_Entry(P1);  // entry action
    ManualStep_Action(N);  // step action
END_STEP
TRANSITION FROM ManualStep TO StopMan
    := NOT xActManual;
END_TRANSITION
STEP StopMan:
    StopMan_Entry(P1);  // entry action
    StopMan_Action(N);  // step action
END_STEP
TRANSITION FROM StopMan TO ModeSelect
    := xExitStop;
END_TRANSITION
TRANSITION FROM ModeSelect TO JogMachineStep
    := xActJogMachine;
END_TRANSITION
STEP JogMachineStep:
    JogMachineStep_Entry(P1);  // entry action
    JogMachineStep_Action(N);  // step action
END_STEP
TRANSITION FROM JogMachineStep TO StopJog
    := NOT xActJogMachine;
END_TRANSITION
STEP StopJog:
    StopJog_Entry(P1);  // entry action
    StopJog_Action(N);  // step action
END_STEP
TRANSITION FROM StopJog TO ModeSelect
    := xExitStop;
END_TRANSITION
TRANSITION FROM ModeSelect TO BrakeReleaseStep
    := xActBrake;
END_TRANSITION
STEP BrakeReleaseStep:
    BrakeReleaseStep_Entry(P1);  // entry action
    BrakeReleaseStep_Action(N);  // step action
END_STEP
TRANSITION FROM BrakeReleaseStep TO StopBrake
    := NOT xActBrake;
END_TRANSITION
STEP StopBrake:
    StopBrake_Entry(P1);  // entry action
    StopBrake_Action(N);  // step action
END_STEP
TRANSITION FROM StopBrake TO ModeSelect
    := xExitStop;
END_TRANSITION
STEP Logic:
    Logic_active(N);  // step action
END_STEP
STEP ExceptionControl:
    ExceptionControl_Action(N);  // step action
END_STEP
STEP Logger:
    Logger_Action(N);  // step action
END_STEP
STEP SubModules:
    SubModules_Action(N);  // step action
END_STEP
STEP Output:
    Output_Action(N);  // step action
END_STEP
TRANSITION FROM (Input, Logic, ExceptionControl, Logger, SubModules, Output) TO Start
    := FALSE;
END_TRANSITION

ACTION _aStart_active:
(* This step is active until the machine is being enabled *)

(* System generated code, do not change without consulting 'Schneider Electric Automation GmbH' - otherwise you risk instability!!!*)
	xVirtualSystem := TPL.FC_GetVirtualSystem();
	
	stMachineInterface.q_sModuleTypeName	:= c_sModuleTypeName;
	stMachineInterface.q_dwModuleType		:= c_dwModuleType;
	stMachineInterface.q_udiModuleVersion	:= c_udiModuleVersion;
(* End of system generated code, do not change without consulting 'Schneider Electric Automation GmbH' - otherwise you risk instability!!!*)

(* System generated code, could be modified for your application *)
	IF(SYSTEMINTERFACE.FC_GetPacDriveBootState() <> 1) THEN
		(* avoid starting as long as the boot of the controller is not finished *)
		stMachineInterface.i_xEnable	:= FALSE; (* set transition condition to FALSE ==> ensure that this step stays active *)

		stMachineInterface.q_etDiag		:= GD.ET_Diag.Ok;
		stMachineInterface.q_udiDiagExt	:= ET_DiagExt.WaitUntilControllerFinishedBoot;
		stMachineInterface.q_sDiagExt	:= FC_EtDiagExtToString(stMachineInterface.q_udiDiagExt);
		stMachineInterface.q_sMsg		:= '';
	ELSE
		stMachineInterface.i_xEnable	:= TRUE;
	END_IF
(* End of system generated code, could be modified for your application *)

(* Application specific code *)
(* ToDo: Add your application specific code here *)
;
(* End of application specific code *)
END_ACTION

ACTION AutoStep_Action:
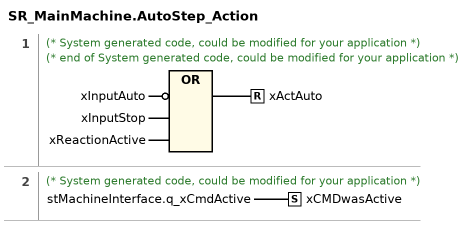
// NETWORK 1
// 					(* System generated code, could be modified for your application *)
// (* end of System generated code, could be modified for your application *)
//
xActAuto R= NOT xInputAuto OR xInputStop OR xReactionActive;

// NETWORK 2
// (* System generated code, could be modified for your application *)
xCMDwasActive S= stMachineInterface.q_xCmdActive;
END_ACTION

ACTION AutoStep_Entry:
(* System generated code, could be modified for your application *)
	xCmdWasActive := FALSE;
	stMachineInterface.iq_diCmd := ET_Cmd.Auto;
(* End of system generated code, could be modified for your application *)
END_ACTION

ACTION AutoStop_Action:
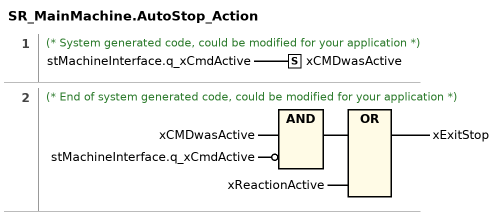
// NETWORK 1
// (* System generated code, could be modified for your application *)
xCMDwasActive S= stMachineInterface.q_xCmdActive;

// NETWORK 2
// (* End of system generated code, could be modified for your application *)
xExitStop := xCMDwasActive AND NOT stMachineInterface.q_xCmdActive OR xReactionActive;
END_ACTION

ACTION AutoStop_Entry:
(* System generated code, could be modified for your application *)
	xCMDwasActive:=FALSE;
	IF	xReactionActive	THEN
		;
	ELSIF stMachineInterface.q_xCmdDone AND NOT stMachineInterface.q_xCmdActive THEN
		stMachineInterface.iq_diCmd := ET_Cmd.Hold;
	ELSE
		stMachineInterface.iq_diCmd := ET_Cmd.Abort;
	END_IF
(* End of system generated code, could be modified for your application *)
END_ACTION

ACTION BrakeReleaseStep_Action:
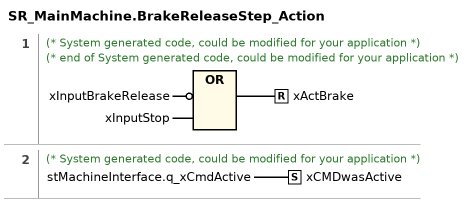
// NETWORK 1
// 					(* System generated code, could be modified for your application *)
// (* end of System generated code, could be modified for your application *)
//
xActBrake R= NOT xInputBrakeRelease OR xInputStop;

// NETWORK 2
// (* System generated code, could be modified for your application *)
xCMDwasActive S= stMachineInterface.q_xCmdActive;
END_ACTION

ACTION BrakeReleaseStep_Entry:
(* System generated code, could be modified for your application *)
	xCMDwasActive		:= FALSE;
	stMachineInterface.iq_diCmd	:= ET_Cmd.BrakeRelease;
(* End of system generated code, could be modified for your application *)
END_ACTION

ACTION ExceptionControl_Action:
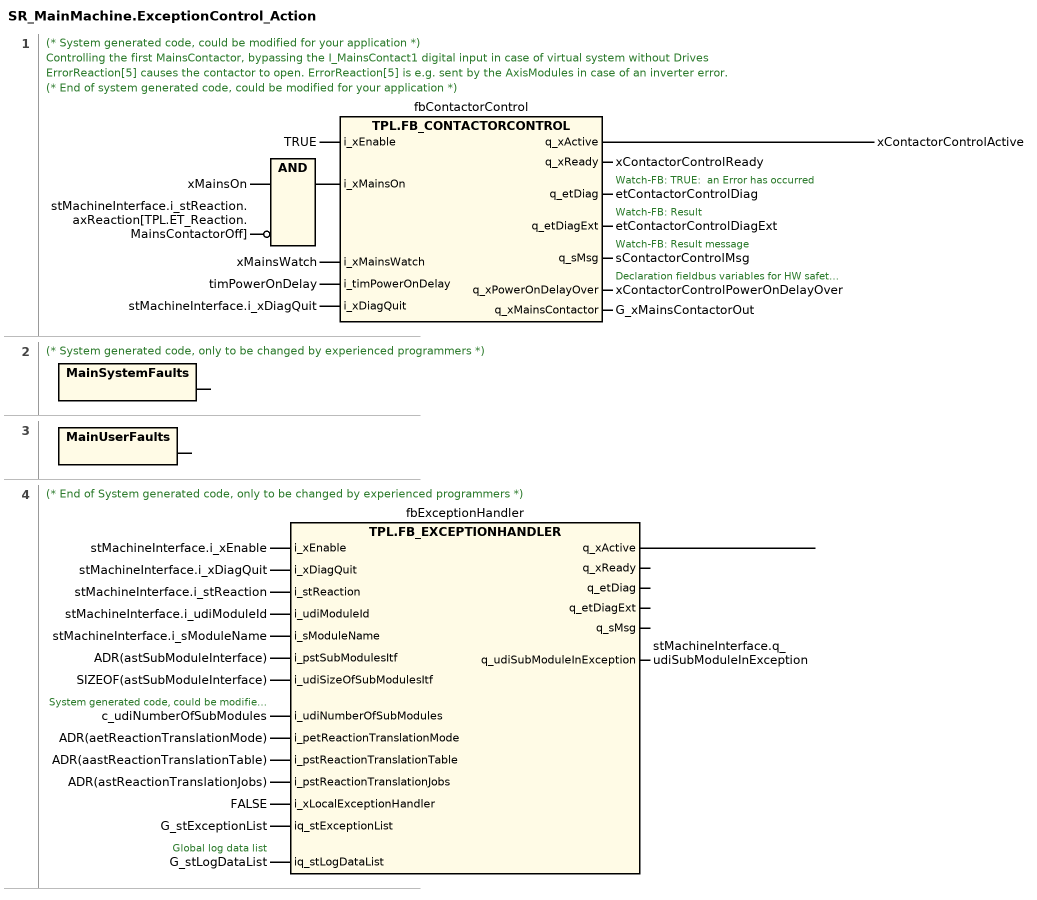
// NETWORK 1
// 					(* System generated code, could be modified for your application *)
// Controlling the first MainsContactor, bypassing the I_MainsContact1 digital input in case of virtual system without Drives
// ErrorReaction[5] causes the contactor to open. ErrorReaction[5] is e.g. sent by the AxisModules in case of an inverter error.
// (* End of system generated code, could be modified for your application *)
//
//   fbContactorControl: Contactor Control related variables
//   etContactorControlDiag: Watch-FB: TRUE: an Error has occurred
//   etContactorControlDiagExt: Watch-FB: Result
//   sContactorControlMsg: Watch-FB: Result message
//   xContactorControlPowerOnDelayOver: Declaration fieldbus variables for HW safety circuit
fbContactorControl(
    i_xEnable := TRUE,
    i_xMainsOn := xMainsOn AND NOT stMachineInterface.i_stReaction.axReaction[TPL.ET_Reaction.MainsContactorOff],
    i_xMainsWatch := xMainsWatch,
    i_timPowerOnDelay := timPowerOnDelay,
    i_xDiagQuit := stMachineInterface.i_xDiagQuit,
    q_xReady => xContactorControlReady,
    q_etDiag => etContactorControlDiag,
    q_etDiagExt => etContactorControlDiagExt,
    q_sMsg => sContactorControlMsg,
    q_xPowerOnDelayOver => xContactorControlPowerOnDelayOver,
    q_xMainsContactor => G_xMainsContactorOut); // TPL.FB_CONTACTORCONTROL
xContactorControlActive := fbContactorControl.q_xActive;

// NETWORK 2
// (* System generated code, only to be changed by experienced programmers *)
MainSystemFaults();

// NETWORK 3
MainUserFaults();

// NETWORK 4
// (* End of System generated code, only to be changed by experienced programmers *)
//   fbExceptionHandler: ExceptionHandling related variables
//   c_udiNumberOfSubModules: System generated code, could be modified for your application
//   G_stLogDataList: Global log data list
fbExceptionHandler(
    i_xEnable := stMachineInterface.i_xEnable,
    i_xDiagQuit := stMachineInterface.i_xDiagQuit,
    i_stReaction := stMachineInterface.i_stReaction,
    i_udiModuleId := stMachineInterface.i_udiModuleId,
    i_sModuleName := stMachineInterface.i_sModuleName,
    i_pstSubModulesItf := ADR(astSubModuleInterface),
    i_udiSizeOfSubModulesItf := SIZEOF(astSubModuleInterface),
    i_udiNumberOfSubModules := c_udiNumberOfSubModules,
    i_petReactionTranslationMode := ADR(aetReactionTranslationMode),
    i_pstReactionTranslationTable := ADR(aastReactionTranslationTable),
    i_pstReactionTranslationJobs := ADR(astReactionTranslationJobs),
    i_xLocalExceptionHandler := FALSE,
    iq_stExceptionList := G_stExceptionList,
    iq_stLogDataList := G_stLogDataList,
    q_udiSubModuleInException => stMachineInterface.q_udiSubModuleInException); // TPL.FB_EXCEPTIONHANDLER
END_ACTION

ACTION Init_Alpha:
(* System generated code, could be modified for your application *)

(* AlphaModule *)
astSubModuleInterface[c_udiAlpha].i_sModuleName		:= STANDARD.CONCAT(STR1 := stMachineInterface.i_sModuleName, STR2 := ': Alpha');
astSubModuleInterface[c_udiAlpha].i_xLogEnable		:= TRUE;
astSubModuleInterface[c_udiAlpha].i_wLogDataFilter	:= UDINT_TO_WORD(TPL.ET_LogDataFilter.ModuleDefault);

(* End of system generated code, could be modified for your application *)
END_ACTION

ACTION Init_Bravo:
(* System generated code, could be modified for your application *)

(* BravoModule *)
astSubModuleInterface[c_udiBravo].i_sModuleName		:= STANDARD.CONCAT(STR1 := stMachineInterface.i_sModuleName, STR2 := ': Bravo');
astSubModuleInterface[c_udiBravo].i_xLogEnable		:= TRUE;
astSubModuleInterface[c_udiBravo].i_wLogDataFilter	:= UDINT_TO_WORD(TPL.ET_LogDataFilter.ModuleDefault);

(* End of system generated code, could be modified for your application *)
END_ACTION

ACTION Init_Charly:
(* System generated code, could be modified for your application *)

(* CharlyModule *)
astSubModuleInterface[c_udiCharly].i_sModuleName	:= STANDARD.CONCAT(STR1 := stMachineInterface.i_sModuleName, STR2 := ': Charly');
astSubModuleInterface[c_udiCharly].i_xLogEnable		:= TRUE;
astSubModuleInterface[c_udiCharly].i_wLogDataFilter	:= UDINT_TO_WORD(TPL.ET_LogDataFilter.ModuleDefault);

(* End of system generated code, could be modified for your application *)
END_ACTION

ACTION Init_CmdTables:
(* System generated code, could be modified for your application *)

(*********************************************************************************************************************)
(*** Prepare  ***)

TPL.FC_FirstStep(udiStepIndex, diStep);
astPrepareTable[udiStepIndex].sTitle					:= 'Prepare AllSubModules';
astPrepareTable[udiStepIndex].udiModuleName				:= TPL.Gc_udiAllSubModules;
astPrepareTable[udiStepIndex].diStep					:= diStep;
astPrepareTable[udiStepIndex].diCMD						:= ET_Cmd.Prepare;
astPrepareTable[udiStepIndex].timTimeOut				:= T#0MS;
astPrepareTable[udiStepIndex].xEndCMD					:= FALSE;

TPL.FC_LastStep(udiStepIndex, diStep);
astPrepareTable[udiStepIndex].sTitle					:= 'End';
astPrepareTable[udiStepIndex].udiModuleName				:= 0;
astPrepareTable[udiStepIndex].diStep					:= diStep;
astPrepareTable[udiStepIndex].diCMD						:= 0;
astPrepareTable[udiStepIndex].timTimeOut				:= T#0MS;
astPrepareTable[udiStepIndex].xEndCMD					:= TRUE;

TPL.FC_FirstCmdTable(iq_udiTableIndex:= udiTableIndex);
astListofCMDTables[udiTableIndex].diCMD					:= ET_Cmd.Prepare;
astListofCMDTables[udiTableIndex].sTitle				:= 'Prepare';
astListofCMDTables[udiTableIndex].udiNumberOfCmdSteps	:= udiStepIndex;

(*********************************************************************************************************************)
(*** Auto  ***)

TPL.FC_FirstStep(udiStepIndex, diStep);
astAutoTable[udiStepIndex].sTitle						:= 'Auto Bravo';
astAutoTable[udiStepIndex].udiModuleName				:= c_udiBravo;
astAutoTable[udiStepIndex].diStep						:= diStep;
astAutoTable[udiStepIndex].diCMD						:= ET_Cmd.Auto;
astAutoTable[udiStepIndex].timTimeOut					:= T#0MS;
astAutoTable[udiStepIndex].xEndCMD						:= FALSE;

TPL.FC_NextStep(udiStepIndex, diStep);
astAutoTable[udiStepIndex].sTitle						:= 'Auto Charly';
astAutoTable[udiStepIndex].udiModuleName				:= c_udiCharly;
astAutoTable[udiStepIndex].diStep						:= diStep;
astAutoTable[udiStepIndex].diCMD						:= ET_Cmd.Auto;
astAutoTable[udiStepIndex].timTimeOut					:= T#0MS;
astAutoTable[udiStepIndex].xEndCMD						:= FALSE;

TPL.FC_NextStep(udiStepIndex, diStep);
astAutoTable[udiStepIndex].sTitle						:= 'Auto Alpha';
astAutoTable[udiStepIndex].udiModuleName				:= c_udiAlpha;
astAutoTable[udiStepIndex].diStep						:= diStep;
astAutoTable[udiStepIndex].diCMD						:= ET_Cmd.Auto;
astAutoTable[udiStepIndex].timTimeOut					:= T#0MS;
astAutoTable[udiStepIndex].xEndCMD						:= FALSE;

TPL.FC_LastStep(udiStepIndex, diStep);
astAutoTable[udiStepIndex].sTitle						:= 'End';
astAutoTable[udiStepIndex].udiModuleName				:= 0;
astAutoTable[udiStepIndex].diStep						:= diStep;
astAutoTable[udiStepIndex].diCMD						:= 0;
astAutoTable[udiStepIndex].timTimeOut					:= T#0MS;
astAutoTable[udiStepIndex].xEndCMD						:= TRUE;

TPL.FC_NextCmdTable(iq_udiTableIndex:= udiTableIndex);
astListofCMDTables[udiTableIndex].diCMD					:= ET_Cmd.Auto;
astListofCMDTables[udiTableIndex].sTitle				:= 'Auto';
astListofCMDTables[udiTableIndex].udiNumberOfCmdSteps	:= udiStepIndex;

(*********************************************************************************************************************)
(*** Manual  ***)

TPL.FC_FirstStep(udiStepIndex, diStep);
astManualTable[udiStepIndex].sTitle						:= 'Stop AllSubModules';
astManualTable[udiStepIndex].udiModuleName				:= TPL.Gc_udiAllSubModules;
astManualTable[udiStepIndex].diStep						:= diStep;
astManualTable[udiStepIndex].diCMD						:= ET_Cmd.Stop;
astManualTable[udiStepIndex].timTimeOut					:= T#0MS;
astManualTable[udiStepIndex].xEndCMD					:= FALSE;

TPL.FC_NextStep(udiStepIndex, diStep);
astManualTable[udiStepIndex].sTitle						:= 'Manual SlaveGroup';
astManualTable[udiStepIndex].udiModuleName				:= c_udiSlaveGroup;
astManualTable[udiStepIndex].diStep						:= diStep;
astManualTable[udiStepIndex].diCMD						:= ET_Cmd.Manual;
astManualTable[udiStepIndex].timTimeOut					:= T#0MS;
astManualTable[udiStepIndex].xEndCMD					:= FALSE;

TPL.FC_LastStep(udiStepIndex, diStep);
astManualTable[udiStepIndex].sTitle						:= 'End';
astManualTable[udiStepIndex].udiModuleName				:= 0;
astManualTable[udiStepIndex].diStep						:= diStep;
astManualTable[udiStepIndex].diCMD						:= 0;
astManualTable[udiStepIndex].timTimeOut					:= T#0MS;
astManualTable[udiStepIndex].xEndCMD					:= TRUE;

TPL.FC_NextCmdTable(iq_udiTableIndex:= udiTableIndex);
astListofCMDTables[udiTableIndex].diCMD					:= ET_Cmd.Manual;
astListofCMDTables[udiTableIndex].sTitle				:= 'Manual';
astListofCMDTables[udiTableIndex].udiNumberOfCmdSteps	:= udiStepIndex;

(*********************************************************************************************************************)
(*** Stop ***)

TPL.FC_FirstStep(udiStepIndex, diStep);
astStopTable[udiStepIndex].sTitle						:= 'Stop AllSubModules';
astStopTable[udiStepIndex].udiModuleName				:= TPL.Gc_udiAllSubModules;
astStopTable[udiStepIndex].diStep						:= diStep;
astStopTable[udiStepIndex].diCMD						:= ET_Cmd.Stop;
astStopTable[udiStepIndex].timTimeOut					:= T#0MS;
astStopTable[udiStepIndex].xEndCMD						:= FALSE;

TPL.FC_LastStep(udiStepIndex, diStep);
astStopTable[udiStepIndex].sTitle						:= 'End';
astStopTable[udiStepIndex].udiModuleName				:= 0;
astStopTable[udiStepIndex].diStep						:= diStep;
astStopTable[udiStepIndex].diCMD						:= 0;
astStopTable[udiStepIndex].timTimeOut					:= T#0MS;
astStopTable[udiStepIndex].xEndCMD						:= TRUE;

TPL.FC_NextCmdTable(iq_udiTableIndex:= udiTableIndex);
astListofCMDTables[udiTableIndex].diCMD					:= ET_Cmd.Stop;
astListofCMDTables[udiTableIndex].sTitle				:= 'Stop';
astListofCMDTables[udiTableIndex].udiNumberOfCmdSteps	:= udiStepIndex;

(*********************************************************************************************************************)
(*** Start ***)

TPL.FC_FirstStep(udiStepIndex, diStep);
astStartTable[udiStepIndex].sTitle						:= 'Start AllSubModules';
astStartTable[udiStepIndex].udiModuleName				:= TPL.Gc_udiAllSubModules;
astStartTable[udiStepIndex].diStep						:= diStep;
astStartTable[udiStepIndex].diCMD						:= ET_Cmd.Start;
astStartTable[udiStepIndex].timTimeOut					:= T#0MS;
astStartTable[udiStepIndex].xEndCMD						:= FALSE;

TPL.FC_LastStep(udiStepIndex, diStep);
astStartTable[udiStepIndex].sTitle						:= 'End';
astStartTable[udiStepIndex].udiModuleName				:= 0;
astStartTable[udiStepIndex].diStep						:= diStep;
astStartTable[udiStepIndex].diCMD						:= 0;
astStartTable[udiStepIndex].timTimeOut					:= T#0MS;
astStartTable[udiStepIndex].xEndCMD						:= TRUE;

TPL.FC_NextCmdTable(iq_udiTableIndex:= udiTableIndex);
astListofCMDTables[udiTableIndex].diCMD					:= ET_Cmd.Start;
astListofCMDTables[udiTableIndex].sTitle				:= 'Start';
astListofCMDTables[udiTableIndex].udiNumberOfCmdSteps	:= udiStepIndex;

(*********************************************************************************************************************)
(*** Abort ***)

TPL.FC_FirstStep(udiStepIndex, diStep);
astAbortTable[udiStepIndex].sTitle						:= 'Abort AllSubModules';
astAbortTable[udiStepIndex].udiModuleName				:= TPL.Gc_udiAllSubModules;
astAbortTable[udiStepIndex].diStep						:= diStep;
astAbortTable[udiStepIndex].diCMD						:= ET_Cmd.Abort;
astAbortTable[udiStepIndex].timTimeOut					:= T#0MS;
astAbortTable[udiStepIndex].xEndCMD						:= FALSE;

TPL.FC_LastStep(udiStepIndex, diStep);
astAbortTable[udiStepIndex].sTitle						:= 'End';
astAbortTable[udiStepIndex].udiModuleName				:= 0;
astAbortTable[udiStepIndex].diStep						:= diStep;
astAbortTable[udiStepIndex].diCMD						:= 0;
astAbortTable[udiStepIndex].timTimeOut					:= T#0MS;
astAbortTable[udiStepIndex].xEndCMD						:= TRUE;

TPL.FC_NextCmdTable(iq_udiTableIndex:= udiTableIndex);
astListofCMDTables[udiTableIndex].diCMD					:= ET_Cmd.Abort;
astListofCMDTables[udiTableIndex].sTitle				:= 'Abort';
astListofCMDTables[udiTableIndex].udiNumberOfCmdSteps	:= udiStepIndex;

(*********************************************************************************************************************)
(*** Hold ***)

TPL.FC_FirstStep(udiStepIndex, diStep);
astHoldTable[udiStepIndex].sTitle						:= 'Hold Alpha';
astHoldTable[udiStepIndex].udiModuleName				:= c_udiAlpha;
astHoldTable[udiStepIndex].diStep						:= diStep;
astHoldTable[udiStepIndex].diCMD						:= ET_Cmd.Hold;
astHoldTable[udiStepIndex].timTimeOut					:= T#0MS;
astHoldTable[udiStepIndex].xEndCMD						:= FALSE;

TPL.FC_NextStep(udiStepIndex, diStep);
astHoldTable[udiStepIndex].sTitle						:= 'Hold Charly';
astHoldTable[udiStepIndex].udiModuleName				:= c_udiCharly;
astHoldTable[udiStepIndex].diStep						:= diStep;
astHoldTable[udiStepIndex].diCMD						:= ET_Cmd.Hold;
astHoldTable[udiStepIndex].timTimeOut					:= T#0MS;
astHoldTable[udiStepIndex].xEndCMD						:= FALSE;

TPL.FC_NextStep(udiStepIndex, diStep);
astHoldTable[udiStepIndex].sTitle						:= 'Hold NodeWithoutMotion';
astHoldTable[udiStepIndex].udiModuleName				:= c_udiNodeWithoutMotion;
astHoldTable[udiStepIndex].diStep						:= diStep;
astHoldTable[udiStepIndex].diCMD						:= ET_Cmd.Hold;
astHoldTable[udiStepIndex].timTimeOut					:= T#0MS;
astHoldTable[udiStepIndex].xEndCMD						:= FALSE;

TPL.FC_LastStep(udiStepIndex, diStep);
astHoldTable[udiStepIndex].sTitle						:= 'End';
astHoldTable[udiStepIndex].udiModuleName				:= 0;
astHoldTable[udiStepIndex].diStep						:= diStep;
astHoldTable[udiStepIndex].diCMD						:= 0;
astHoldTable[udiStepIndex].timTimeOut					:= T#0MS;
astHoldTable[udiStepIndex].xEndCMD						:= TRUE;

TPL.FC_NextCmdTable(iq_udiTableIndex:= udiTableIndex);
astListofCMDTables[udiTableIndex].diCMD					:= ET_Cmd.Hold;
astListofCMDTables[udiTableIndex].sTitle				:= 'Hold';
astListofCMDTables[udiTableIndex].udiNumberOfCmdSteps	:= udiStepIndex;

(*********************************************************************************************************************)
(*** Hold for JogMachine***)

TPL.FC_FirstStep(udiStepIndex, diStep);
astHoldJogMachineTable[udiStepIndex].sTitle				:= 'Stop Alpha';
astHoldJogMachineTable[udiStepIndex].udiModuleName		:= c_udiAlpha;
astHoldJogMachineTable[udiStepIndex].diStep				:= diStep;
astHoldJogMachineTable[udiStepIndex].diCMD				:= ET_Cmd.Stop;
astHoldJogMachineTable[udiStepIndex].timTimeOut			:= T#0MS;
astHoldJogMachineTable[udiStepIndex].xEndCMD			:= FALSE;

TPL.FC_NextStep(udiStepIndex, diStep);
astHoldJogMachineTable[udiStepIndex].sTitle				:= 'Hold Charly';
astHoldJogMachineTable[udiStepIndex].udiModuleName		:= c_udiCharly;
astHoldJogMachineTable[udiStepIndex].diStep				:= diStep;
astHoldJogMachineTable[udiStepIndex].diCMD				:= ET_Cmd.Hold;
astHoldJogMachineTable[udiStepIndex].timTimeOut			:= T#0MS;
astHoldJogMachineTable[udiStepIndex].xEndCMD			:= FALSE;

TPL.FC_NextStep(udiStepIndex, diStep);
astHoldJogMachineTable[udiStepIndex].sTitle				:= 'Hold NodeWithoutMotion';
astHoldJogMachineTable[udiStepIndex].udiModuleName		:= c_udiNodeWithoutMotion;
astHoldJogMachineTable[udiStepIndex].diStep				:= diStep;
astHoldJogMachineTable[udiStepIndex].diCMD				:= ET_Cmd.Hold;
astHoldJogMachineTable[udiStepIndex].timTimeOut			:= T#0MS;
astHoldJogMachineTable[udiStepIndex].xEndCMD			:= FALSE;

TPL.FC_LastStep(udiStepIndex, diStep);
astHoldJogMachineTable[udiStepIndex].sTitle				:= 'End';
astHoldJogMachineTable[udiStepIndex].udiModuleName		:= 0;
astHoldJogMachineTable[udiStepIndex].diStep				:= diStep;
astHoldJogMachineTable[udiStepIndex].diCMD				:= 0;
astHoldJogMachineTable[udiStepIndex].timTimeOut			:= T#0MS;
astHoldJogMachineTable[udiStepIndex].xEndCMD			:= TRUE;

TPL.FC_NextCmdTable(iq_udiTableIndex:= udiTableIndex);
astListofCMDTables[udiTableIndex].diCMD					:= ET_Cmd.HoldJM;
astListofCMDTables[udiTableIndex].sTitle				:= 'Hold Jog Machine';
astListofCMDTables[udiTableIndex].udiNumberOfCmdSteps	:= udiStepIndex;

(*********************************************************************************************************************)
(*** Brake Release ***)

TPL.FC_FirstStep(udiStepIndex, diStep);
astBrakeReleaseTable[udiStepIndex].sTitle				:= 'BrakeRelease Bravo';
astBrakeReleaseTable[udiStepIndex].udiModuleName		:= c_udiBravo;
astBrakeReleaseTable[udiStepIndex].diStep				:= diStep;
astBrakeReleaseTable[udiStepIndex].diCMD				:= ET_Cmd.BrakeRelease;
astBrakeReleaseTable[udiStepIndex].timTimeOut			:= T#0MS;
astBrakeReleaseTable[udiStepIndex].xEndCMD				:= FALSE;

TPL.FC_LastStep(udiStepIndex, diStep);
astBrakeReleaseTable[udiStepIndex].sTitle				:= 'End';
astBrakeReleaseTable[udiStepIndex].udiModuleName		:= 0;
astBrakeReleaseTable[udiStepIndex].diStep				:= diStep;
astBrakeReleaseTable[udiStepIndex].diCMD				:= 0;
astBrakeReleaseTable[udiStepIndex].timTimeOut			:= T#0MS;
astBrakeReleaseTable[udiStepIndex].xEndCMD				:= TRUE;

TPL.FC_NextCmdTable(iq_udiTableIndex:= udiTableIndex);
astListofCMDTables[udiTableIndex].diCMD					:= ET_Cmd.BrakeRelease;
astListofCMDTables[udiTableIndex].sTitle				:= 'BrakeRelease';
astListofCMDTables[udiTableIndex].udiNumberOfCmdSteps	:= udiStepIndex;

(*********************************************************************************************************************)
(*** JogMachine ***)

TPL.FC_FirstStep(udiStepIndex, diStep);
astJogMachineTable[udiStepIndex].sTitle					:= 'Auto Bravo';
astJogMachineTable[udiStepIndex].udiModuleName			:= c_udiBravo;
astJogMachineTable[udiStepIndex].diStep					:= diStep;
astJogMachineTable[udiStepIndex].diCMD					:= ET_Cmd.Auto;
astJogMachineTable[udiStepIndex].timTimeOut				:= T#0MS;
astJogMachineTable[udiStepIndex].xEndCMD				:= FALSE;

TPL.FC_NextStep(udiStepIndex, diStep);
astJogMachineTable[udiStepIndex].sTitle					:= 'Auto Charly';
astJogMachineTable[udiStepIndex].udiModuleName			:= c_udiCharly;
astJogMachineTable[udiStepIndex].diStep					:= diStep;
astJogMachineTable[udiStepIndex].diCMD					:= ET_Cmd.Auto;
astJogMachineTable[udiStepIndex].timTimeOut				:= T#0MS;
astJogMachineTable[udiStepIndex].xEndCMD				:= FALSE;

TPL.FC_NextStep(udiStepIndex, diStep);
astJogMachineTable[udiStepIndex].sTitle					:= 'Manual Alpha';
astJogMachineTable[udiStepIndex].udiModuleName			:= c_udiAlpha;
astJogMachineTable[udiStepIndex].diStep					:= diStep;
astJogMachineTable[udiStepIndex].diCMD					:= ET_Cmd.Manual;
astJogMachineTable[udiStepIndex].timTimeOut				:= T#0MS;
astJogMachineTable[udiStepIndex].xEndCMD				:= FALSE;

TPL.FC_LastStep(udiStepIndex, diStep);
astJogMachineTable[udiStepIndex].sTitle					:= 'End';
astJogMachineTable[udiStepIndex].udiModuleName			:= 0;
astJogMachineTable[udiStepIndex].diStep					:= diStep;
astJogMachineTable[udiStepIndex].diCMD					:= 0;
astJogMachineTable[udiStepIndex].timTimeOut				:= T#0MS;
astJogMachineTable[udiStepIndex].xEndCMD				:= TRUE;

TPL.FC_NextCmdTable(iq_udiTableIndex:= udiTableIndex);
astListofCMDTables[udiTableIndex].diCMD					:= ET_Cmd.Jogging;
astListofCMDTables[udiTableIndex].sTitle				:= 'Jogging';
astListofCMDTables[udiTableIndex].udiNumberOfCmdSteps	:= udiStepIndex;

(* End of system generated code, could be modified for your application *)
END_ACTION

ACTION Init_Exceptions:
(* System generated code, could be modified for your application *)

(*
	TPL.ET_Reaction.AsyncStop
	TPL.ET_Reaction.SyncStopEL
	TPL.ET_Reaction.SyncStopEH
	TPL.ET_Reaction.StopEndOfCycle
	TPL.ET_Reaction.MainsContactorOff
*)

(*------------------------------------------------------------------------------------------*)
(* Init System Exceptions *)
(*------------------------------------------------------------------------------------------*)

stSystemException1.etDiag														:= GD.ET_Diag.Ok; (* Replaced on usage *)
stSystemException1.udiDiagExt													:= ET_DiagExt.Ok; (* Replaced on usage *)
stSystemException1.sDiagExt														:= FC_EtDiagExtToString(ET_DiagExt.Ok); (* Replaced on usage *)
stSystemException1.sMsg															:= ''; (* Replaced on usage *)
stSystemException1.udiModuleId													:= stMachineInterface.i_udiModuleId;
stSystemException1.sModuleName													:= stMachineInterface.i_sModuleName;
stSystemException1.etSource														:= TPL.ET_ExceptionSource.Main;
stSystemException1.timDelayTime													:= T#0MS;
stSystemException1.wHmiAttributes												:= 0;
stSystemException1.xAutoQuit													:= FALSE;
stSystemException1.stReaction.axReaction[TPL.ET_Reaction.AsyncStop]				:= TRUE;

stSystemException2.etDiag														:= GD.ET_Diag.Ok; (* Replaced on usage *)
stSystemException2.udiDiagExt													:= ET_DiagExt.Ok; (* Replaced on usage *)
stSystemException2.sDiagExt														:= FC_EtDiagExtToString(ET_DiagExt.Ok); (* Replaced on usage *)
stSystemException2.sMsg															:= ''; (* Replaced on usage *)
stSystemException2.udiModuleId													:= stMachineInterface.i_udiModuleId;
stSystemException2.sModuleName													:= stMachineInterface.i_sModuleName;
stSystemException2.etSource														:= TPL.ET_ExceptionSource.Main;
stSystemException2.timDelayTime													:= T#0MS;
stSystemException2.wHmiAttributes												:= 0;
stSystemException2.xAutoQuit													:= FALSE;
stSystemException2.stReaction.axReaction[TPL.ET_Reaction.SyncStopEL]			:= TRUE;

stSystemException3.etDiag														:= GD.ET_Diag.Ok; (* Replaced on usage *)
stSystemException3.udiDiagExt													:= ET_DiagExt.Ok; (* Replaced on usage *)
stSystemException3.sDiagExt														:= FC_EtDiagExtToString(ET_DiagExt.Ok); (* Replaced on usage *)
stSystemException3.sMsg															:= ''; (* Replaced on usage *)
stSystemException3.udiModuleId													:= stMachineInterface.i_udiModuleId;
stSystemException3.sModuleName													:= stMachineInterface.i_sModuleName;
stSystemException3.etSource														:= TPL.ET_ExceptionSource.Main;
stSystemException3.timDelayTime													:= T#0MS;
stSystemException3.wHmiAttributes												:= 0;
stSystemException3.xAutoQuit													:= FALSE;
stSystemException3.stReaction.axReaction[TPL.ET_Reaction.SyncStopEH]			:= TRUE;

stEmergencyStopException.etDiag													:= GD.ET_Diag.ExecutionAborted;
stEmergencyStopException.udiDiagExt												:= ET_DiagExt.MainSystemEmergencyStop;
stEmergencyStopException.sDiagExt												:= FC_EtDiagExtToString(ET_DiagExt.MainSystemEmergencyStop);
stEmergencyStopException.sMsg													:= 'Emergency Stop';
stEmergencyStopException.udiModuleId											:= stMachineInterface.i_udiModuleId;
stEmergencyStopException.sModuleName											:= stMachineInterface.i_sModuleName;
stEmergencyStopException.etSource												:= TPL.ET_ExceptionSource.Main;
stEmergencyStopException.timDelayTime											:= T#0MS;
stEmergencyStopException.wHmiAttributes											:= 0;
stEmergencyStopException.xAutoQuit												:= FALSE;
stEmergencyStopException.stReaction.axReaction[TPL.ET_Reaction.SyncStopEL]		:= TRUE;

stContactorControlException.etDiag												:= GD.ET_Diag.Ok; (* Replaced on usage *)
stContactorControlException.udiDiagExt											:= ET_DiagExt.Ok; (* Replaced on usage *)
stContactorControlException.sDiagExt											:= FC_EtDiagExtToString(ET_DiagExt.Ok); (* Replaced on usage *)
stContactorControlException.sMsg												:= ''; (* Replaced on usage *)
stContactorControlException.udiModuleId											:= stMachineInterface.i_udiModuleId;
stContactorControlException.sModuleName											:= stMachineInterface.i_sModuleName;
stContactorControlException.etSource											:= TPL.ET_ExceptionSource.Main;
stContactorControlException.timDelayTime										:= T#0MS;
stContactorControlException.wHmiAttributes										:= 0;
stContactorControlException.xAutoQuit											:= FALSE;
stContactorControlException.stReaction.axReaction[TPL.ET_Reaction.AsyncStop]	:= TRUE;

stUpdateStructsException.etDiag													:= GD.ET_Diag.UnexpectedProgramBehavior;
stUpdateStructsException.udiDiagExt												:= ET_DiagExt.UpdateStructsException;
stUpdateStructsException.sDiagExt												:= FC_EtDiagExtToString(i_etDiagExt := stUpdateStructsException.udiDiagExt);
stUpdateStructsException.sMsg													:= '';	(* Replaced on usage *)
stUpdateStructsException.udiModuleId											:= stMachineInterface.i_udiModuleId;
stUpdateStructsException.sModuleName											:= stMachineInterface.i_sModuleName;
stUpdateStructsException.stReaction.axReaction[TPL.ET_Reaction.AsyncStop]		:= TRUE;
stUpdateStructsException.etSource												:= TPL.ET_ExceptionSource.Main;
stUpdateStructsException.timDelayTime											:= T#0MS;
stUpdateStructsException.wHmiAttributes											:= 0;
stUpdateStructsException.xAutoQuit												:= FALSE;

stInitReactionsException.etDiag													:= GD.ET_Diag.UnexpectedProgramBehavior;
stInitReactionsException.udiDiagExt												:= ET_DiagExt.InitReactionsException;
stInitReactionsException.sDiagExt												:= FC_EtDiagExtToString(i_etDiagExt := stInitReactionsException.udiDiagExt);
stInitReactionsException.sMsg													:= '';	(* Replaced on usage *)
stInitReactionsException.udiModuleId											:= stMachineInterface.i_udiModuleId;
stInitReactionsException.sModuleName											:= stMachineInterface.i_sModuleName;
stInitReactionsException.stReaction.axReaction[TPL.ET_Reaction.AsyncStop]		:= TRUE;
stInitReactionsException.etSource												:= TPL.ET_ExceptionSource.Main;
stInitReactionsException.timDelayTime											:= T#0MS;
stInitReactionsException.wHmiAttributes											:= 0;
stInitReactionsException.xAutoQuit												:= FALSE;

stInitSubModulesException.etDiag												:= GD.ET_Diag.UnexpectedProgramBehavior;
stInitSubModulesException.udiDiagExt											:= ET_DiagExt.InitSubModulesException;
stInitSubModulesException.sDiagExt												:= FC_EtDiagExtToString(i_etDiagExt := stInitSubModulesException.udiDiagExt);
stInitSubModulesException.sMsg													:= '';	(* Replaced on usage *)
stInitSubModulesException.udiModuleId											:= stMachineInterface.i_udiModuleId;
stInitSubModulesException.sModuleName											:= stMachineInterface.i_sModuleName;
stInitSubModulesException.stReaction.axReaction[TPL.ET_Reaction.AsyncStop]		:= TRUE;
stInitSubModulesException.etSource												:= TPL.ET_ExceptionSource.Main;
stInitSubModulesException.timDelayTime											:= T#0MS;
stInitSubModulesException.wHmiAttributes										:= 0;
stInitSubModulesException.xAutoQuit												:= FALSE;

(*------------------------------------------------------------------------------------------*)
(* Init User Exceptions *)
(*------------------------------------------------------------------------------------------*)	

stUserException1.etDiag															:= GD.ET_Diag.ExecutionAborted; (* Replaced on usage *)
stUserException1.udiDiagExt														:= ET_DiagExtUser.Exception1FromMain; (* Replaced on usage *)
stUserException1.sDiagExt														:= FC_EtDiagExtUserToString(i_etDiagExt := stUserException1.udiDiagExt); (* Replaced on usage *)
stUserException1.sMsg															:= 'User Exception 1'; (* To be replaced if used *)
stUserException1.udiModuleId													:= stMachineInterface.i_udiModuleId;
stUserException1.sModuleName													:= stMachineInterface.i_sModuleName;
stUserException1.etSource														:= TPL.ET_ExceptionSource.User;
stUserException1.timDelayTime													:= T#0MS;
stUserException1.wHmiAttributes													:= 0;
stUserException1.xAutoQuit														:= FALSE;
stUserException1.stReaction.axReaction[TPL.ET_Reaction.AsyncStop]				:= TRUE;

stUserException2.etDiag															:= GD.ET_Diag.ExecutionAborted; (* Replaced on usage *)
stUserException2.udiDiagExt														:= ET_DiagExtUser.Exception2FromMain; (* Replaced on usage *)
stUserException2.sDiagExt														:= FC_EtDiagExtUserToString(i_etDiagExt := stUserException2.udiDiagExt); (* Replaced on usage *)
stUserException2.sMsg															:= 'User Exception 2'; (* To be replaced if used *)
stUserException2.udiModuleId													:= stMachineInterface.i_udiModuleId;
stUserException2.sModuleName													:= stMachineInterface.i_sModuleName;
stUserException2.etSource														:= TPL.ET_ExceptionSource.User;
stUserException2.timDelayTime													:= T#0MS;
stUserException2.wHmiAttributes													:= 0;
stUserException2.xAutoQuit														:= FALSE;
stUserException2.stReaction.axReaction[TPL.ET_Reaction.SyncStopEL]				:= TRUE;

stUserException3.etDiag															:= GD.ET_Diag.ExecutionAborted; (* Replaced on usage *)
stUserException3.udiDiagExt														:= ET_DiagExtUser.Exception3FromMain; (* Replaced on usage *)
stUserException3.sDiagExt														:= FC_EtDiagExtUserToString(i_etDiagExt := stUserException3.udiDiagExt); (* Replaced on usage *)
stUserException3.sMsg															:= 'User Exception 3'; (* To be replaced if used *)
stUserException3.udiModuleId													:= stMachineInterface.i_udiModuleId;
stUserException3.sModuleName													:= stMachineInterface.i_sModuleName;
stUserException3.etSource														:= TPL.ET_ExceptionSource.User;
stUserException3.timDelayTime													:= T#0MS;
stUserException3.wHmiAttributes													:= 0;
stUserException3.xAutoQuit														:= TRUE;
stUserException3.stReaction.axReaction[TPL.ET_Reaction.SyncStopEH]				:= TRUE;

stUserException4.etDiag															:= GD.ET_Diag.ExecutionAborted; (* Replaced on usage *)
stUserException4.udiDiagExt														:= ET_DiagExtUser.Exception4FromMain; (* Replaced on usage *)
stUserException4.sDiagExt														:= FC_EtDiagExtUserToString(i_etDiagExt := stUserException4.udiDiagExt); (* Replaced on usage *)
stUserException4.sMsg															:= 'User Exception 4'; (* To be replaced if used *)	
stUserException4.udiModuleId													:= stMachineInterface.i_udiModuleId;
stUserException4.sModuleName													:= stMachineInterface.i_sModuleName;
stUserException4.etSource														:= TPL.ET_ExceptionSource.User;
stUserException4.timDelayTime													:= T#0MS;
stUserException4.wHmiAttributes													:= 0;
stUserException4.xAutoQuit														:= FALSE;
stUserException4.stReaction.axReaction[TPL.ET_Reaction.StopEndOfCycle]			:= TRUE;

stUserException5.etDiag															:= GD.ET_Diag.ExecutionAborted; (* Replaced on usage *)
stUserException5.udiDiagExt														:= ET_DiagExtUser.Exception5FromMain; (* Replaced on usage *)
stUserException5.sDiagExt														:= FC_EtDiagExtUserToString(i_etDiagExt := stUserException5.udiDiagExt); (* Replaced on usage *)
stUserException5.sMsg															:= 'User Exception 5'; (* To be replaced if used *)		
stUserException5.udiModuleId													:= stMachineInterface.i_udiModuleId;
stUserException5.sModuleName													:= stMachineInterface.i_sModuleName;
stUserException5.etSource														:= TPL.ET_ExceptionSource.User;
stUserException5.timDelayTime													:= T#0MS;
stUserException5.wHmiAttributes													:= 0;
stUserException5.xAutoQuit														:= FALSE;
stUserException5.stReaction.axReaction[TPL.ET_Reaction.MainsContactorOff]		:= TRUE;
stUserException5.stReaction.axReaction[TPL.ET_Reaction.StopEndOfCycle]			:= TRUE;

(* End of system generated code, could be modified for your application *)
END_ACTION

ACTION Init_NodeWithoutMotion:
(* System generated code, could be modified for your application *)

(* Module NodeWithoutMotion *)
astSubModuleInterface[c_udiNodeWithoutMotion].i_sModuleName		:= STANDARD.CONCAT(STR1 := stMachineInterface.i_sModuleName, STR2 := ': NodeWithoutMotion');
astSubModuleInterface[c_udiNodeWithoutMotion].i_xLogEnable		:= TRUE;
astSubModuleInterface[c_udiNodeWithoutMotion].i_wLogDataFilter	:= UDINT_TO_WORD(TPL.ET_LogDataFilter.ModuleDefault);

(* End of system generated code, could be modified for your application *)
END_ACTION

ACTION Init_Reactions:
(* System generated code, only to be changed by experienced programmers *)
IF c_udiNumberOfSubModules < 1 THEN
	RETURN;
END_IF

(* Change of default reactions only on demand *)

xInitReactionsException := FALSE;

(*****************************************************************************************************************************************************)
(* Init ReactionTranslationMode *)

TPL.FC_InitReactionTranslationMode(	i_udiNumberOfSubModules			:= c_udiNumberOfSubModules,
									i_petReactionTranslationMode	:= ADR(aetReactionTranslationMode),
									q_etDiag						=> etDiag,
									q_etDiagExt						=> etDiagExtTPL);
							
IF etDiag <> GD.ET_Diag.Ok AND NOT xInitReactionsException THEN
	xInitReactionsException := TRUE;
	
	stInitReactionsException.sMsg := PDL.FC_MultiConcat(i_sString1 := 'InitReactionTranslationMode - ', 
														i_sString2 := GD.FC_EtDiagToString(i_etDiag := etDiag), 
														i_sString3 := ' - ', 
														i_sString4 := TPL.FC_EtDiagExtToString(i_etDiagExt := etDiagExtTPL));
END_IF	

(*****************************************************************************************************************************************************)
(* Init ReactionTranslationTable *)	

TPL.FC_InitReactionTranslationTable(i_udiNumberOfSubModules			:= c_udiNumberOfSubModules,
									i_pstReactionTranslationTable	:= ADR(aastReactionTranslationTable),
									q_etDiag						=> etDiag,
									q_etDiagExt						=> etDiagExtTPL);
									
IF etDiag <> GD.ET_Diag.Ok AND NOT xInitReactionsException THEN
	xInitReactionsException := TRUE;
	
	stInitReactionsException.sMsg := PDL.FC_MultiConcat(i_sString1 := 'InitReactionTranslationTable - ', 
														i_sString2 := GD.FC_EtDiagToString(i_etDiag := etDiag), 
														i_sString3 := ' - ', 
														i_sString4 := TPL.FC_EtDiagExtToString(i_etDiagExt := etDiagExtTPL));
END_IF		

(*****************************************************************************************************************************************************)
(* Init ReactionTranslationJobs *)	
								
TPL.FC_InitReactionTranslationJobs( i_udiNumberOfSubModules			:= c_udiNumberOfSubModules,
									i_pstReactionTranslationJobs	:= ADR(astReactionTranslationJobs),
									q_etDiag						=> etDiag,
									q_etDiagExt						=> etDiagExtTPL);
						
IF etDiag <> GD.ET_Diag.Ok AND NOT xInitReactionsException THEN
	xInitReactionsException := TRUE;
	
	stInitReactionsException.sMsg := PDL.FC_MultiConcat(i_sString1 := 'InitReactionTranslationJobs - ', 
														i_sString2 := GD.FC_EtDiagToString(i_etDiag := etDiag), 
														i_sString3 := ' - ', 
														i_sString4 := TPL.FC_EtDiagExtToString(i_etDiagExt := etDiagExtTPL));
END_IF		

(*****************************************************************************************************************************************************)
(* Set exception if any exception occurred *)

TPL.FC_SetException(i_xExceptionActive	:= xInitReactionsException, 
					iq_stException		:= stInitReactionsException, 
					iq_stExceptionList	:= G_stExceptionList, 
					iq_stLogDataList	:= G_stLogDataList);
					
xInitSuccessful := xInitSuccessful AND NOT xInitReactionsException;

etDiag := GD.ET_Diag.Ok;
(* End of system generated code, do not change without consulting 'Schneider Electric Automation GmbH' - otherwise you risk instability!!!*)

(* System generated code, could be modified for your application *)

(* Change of default reactions only if necessary *)
(* Examples: *)

(* A translation mode must be set for each module where the reactions should be translated *)

(* Reaction TPL.ET_Reaction.SyncStopEH in the MainMachine should act as Reaction TPL.ET_Reaction.StopEndOfCycle in BravoModule *)
// aetReactionTranslationMode[c_udiBravo] := TPL.ET_ReactionTranslationMode.Table;
// aastReactionTranslationTable[c_udiBravo,TPL.ET_Reaction.SyncStopEH].axReaction[TPL.ET_Reaction.SyncStopEH]		:= FALSE;	(* Reset old reaction *)
// aastReactionTranslationTable[c_udiBravo,TPL.ET_Reaction.SyncStopEH].axReaction[TPL.ET_Reaction.StopEndOfCycle]	:= TRUE;	(* Set new reaction *)

(* Reaction TPL.ET_Reaction.SyncStopEL in the MainMachine should act as Reaction TPL.ET_Reaction.StopEndOfCycle and TPL.ET_Reaction.MainsContactorOff in CharlyModule *)
// aetReactionTranslationMode[c_udiCharly] := TPL.ET_ReactionTranslationMode.Table;
// aastReactionTranslationTable[c_udiCharly,TPL.ET_Reaction.SyncStopEL].axReaction[TPL.ET_Reaction.SyncStopEL]			:= FALSE;	(* Reset old reaction *)
// aastReactionTranslationTable[c_udiCharly,TPL.ET_Reaction.SyncStopEL].axReaction[TPL.ET_Reaction.StopEndOfCycle]		:= TRUE;	(* Set new reaction *)
// aastReactionTranslationTable[c_udiCharly,TPL.ET_Reaction.SyncStopEL].axReaction[TPL.ET_Reaction.MainsContactorOff]	:= TRUE;	(* Set new reaction *)

(* Reaction TPL.ET_Reaction.SyncStopEL + TPL.ET_Reaction.SyncStopEH + TPL.ET_Reaction.StopEndOfCycle in the MainMachine should act as Reaction TPL.ET_Reaction.AsyncStop in AlphaModule *)
// aetReactionTranslationMode[c_udiBravo] := TPL.ET_ReactionTranslationMode.Table;
// aastReactionTranslationTable[c_udiAlpha,TPL.ET_Reaction.SyncStopEL].axReaction[TPL.ET_Reaction.SyncStopEL]			:= FALSE;	(* Reset old reaction *)
// aastReactionTranslationTable[c_udiAlpha,TPL.ET_Reaction.SyncStopEH].axReaction[TPL.ET_Reaction.SyncStopEH]			:= FALSE;	(* Reset old reaction *)
// aastReactionTranslationTable[c_udiAlpha,TPL.ET_Reaction.StopEndOfCycle].axReaction[TPL.ET_Reaction.StopEndOfCycle]	:= FALSE;	(* Reset old reaction *)
// aastReactionTranslationTable[c_udiAlpha,TPL.ET_Reaction.SyncStopEL].axReaction[TPL.ET_Reaction.AsyncStop]			:= TRUE;	(* Set new reaction *)
// aastReactionTranslationTable[c_udiAlpha,TPL.ET_Reaction.SyncStopEH].axReaction[TPL.ET_Reaction.AsyncStop]			:= TRUE;	(* Set new reaction *)
// aastReactionTranslationTable[c_udiAlpha,TPL.ET_Reaction.StopEndOfCycle].axReaction[TPL.ET_Reaction.AsyncStop]		:= TRUE;	(* Set new reaction *)

(* End of system generated code, could be modified for your application *)
END_ACTION

ACTION Init_SubModules:
(* System generated code, could be modified for your application *)

(* Module Group declaration *)

aaudiSubModuleGroups[c_udiMasterGroup-TPL.Gc_udiGroupOffset,TPL.ET_Group.Member1]	:= c_udiAlpha;		(* The c_udiAlpha is the first element of the group c_udiMasterGroup *)
aaudiSubModuleGroups[c_udiMasterGroup-TPL.Gc_udiGroupOffset,TPL.ET_Group.Member2]	:= 0;				(* There is no second element of the group c_udiMasterGroup *)

aaudiSubModuleGroups[c_udiSlaveGroup-TPL.Gc_udiGroupOffset,TPL.ET_Group.Member1]	:= c_udiBravo;		(* The c_udiBravo is the first element of the group c_udiSlaveGroup *)
aaudiSubModuleGroups[c_udiSlaveGroup-TPL.Gc_udiGroupOffset,TPL.ET_Group.Member2]	:= c_udiCharly;		(* The c_udiCharly is the second element of the group c_udiSlaveGroup *)


(* Configuration of exception logging *)
G_stLogDataList.wExceptionLogDataFilter	:= UDINT_TO_WORD(TPL.ET_LogDataFilter.ExceptionListDefault);

(* Exception in case of an overflow of the exception list - Set ModuleId and ModuleName *)
G_stExceptionList.stOverflowException.udiModuleId	:= stMachineInterface.i_udiModuleId;
G_stExceptionList.stOverflowException.sModuleName	:= stMachineInterface.i_sModuleName;


(* Example, how to modify the reaction of the overflow exception, by default all reactions are set *)
// FC_ReinitReaction(iq_stException := G_stExceptionList.stOverflowError); //set reaction to no reaction
// G_stExceptionList.stOverflowException.stReaction.axReaction[TPL.ET_Reaction.AsyncStop] := TRUE;
// G_stExceptionList.stOverflowException.stReaction.axReaction[TPL.ET_Reaction.MainsContactorOff] := TRUE; //ensure that the worst possible reactions for your machine are set


(* Set logger save file name and path *)
G_stLoggerInterface.i_sFileName		:= 'ram0:TPL_LOG.XML';					(* 'ide0:TPL_LOG.XML', 'ram0:TPL_LOG.CSV', 'remote:ram0:\\TPL_LOG.XML' *)
G_stLoggerInterface.i_xEnable		:= TRUE;
G_stLoggerInterface.i_etSortKey		:= TPL.ET_LogDataSortKey.SortByTime;	(*	TPL.ET_LogDataSortKey.SortByCmd
																				TPL.ET_LogDataSortKey.SortById
																				TPL.ET_LogDataSortKey.SortByModuleId
																				TPL.ET_LogDataSortKey.SortByModuleIdAndTime
																				TPL.ET_LogDataSortKey.SortByName
																				TPL.ET_LogDataSortKey.SortByReaction
																				TPL.ET_LogDataSortKey.SortByTime *)

(* End of system generated code, could be modified for your application *)

(* System generated code, do not change without consulting 'Schneider Electric Automation GmbH' - otherwise you risk instability!!!*)
xInitSubModulesException := FALSE;

(*****************************************************************************************************************************************************)
(* Set IDs of SubModules *)	

TPL.FC_SetSubModuleIds(	i_udiMainModuleID			:= stMachineInterface.i_udiModuleId,
						i_pstSubModulesItf			:= ADR(astSubModuleInterface),
						i_udiNumberOfSubModules		:= c_udiNumberOfSubModules,
						q_etDiag					=> etDiag,
						q_etDiagExt					=> etDiagExtTPL);
					
IF etDiag <> GD.ET_Diag.Ok AND NOT xInitSubModulesException THEN
	xInitSubModulesException := TRUE;
	
	stInitSubModulesException.sMsg := PDL.FC_MultiConcat(	i_sString1 := 'SetSubModuleIds - ', 
															i_sString2 := GD.FC_EtDiagToString(i_etDiag := etDiag), 
															i_sString3 := ' - ', 
															i_sString4 := TPL.FC_EtDiagExtToString(i_etDiagExt := etDiagExtTPL));
END_IF	

(*****************************************************************************************************************************************************)
(* Set exception if any exception occurred *)

TPL.FC_SetException(i_xExceptionActive	:= xInitSubModulesException, 
					iq_stException		:= stInitSubModulesException, 
					iq_stExceptionList	:= G_stExceptionList, 
					iq_stLogDataList	:= G_stLogDataList);

xInitSuccessful := xInitSuccessful AND NOT xInitSubModulesException;
					
etDiag := GD.ET_Diag.Ok;
					
(* End of system generated code, do not change without consulting 'Schneider Electric Automation GmbH' - otherwise you risk instability!!!*)
END_ACTION

ACTION InitModule_Action:
(* This step is used for initialisations after being enabled *)

(* System generated code, do not change without consulting 'Schneider Electric Automation GmbH' - otherwise you risk instability!!!*)
xInitSuccessful := TRUE;

stMachineInterface.q_xActive		:= TRUE;
stMachineInterface.q_xReady			:= FALSE;
stMachineInterface.q_etDiag			:= GD.ET_Diag.Ok;
stMachineInterface.q_udiDiagExt		:= ET_DiagExt.Initializing;
stMachineInterface.q_sDiagExt		:= FC_EtDiagExtToString(i_etDiagExt := ET_DiagExt.Initializing);
stMachineInterface.q_sMsg			:= '';

stMachineInterface.i_sModuleName		:= 'MainMachine';
stMachineInterface.i_udiModuleId		:= c_udiMainModuleId;
stMachineInterface.i_xLogEnable			:= TRUE;
stMachineInterface.i_wLogDataFilter		:= UDINT_TO_WORD(TPL.ET_LogDataFilter.ModuleDefault);

SYSTEMINTERFACE.FC_DiagNoQuitSet(i_diDiagCode := 8316);
(* End of system generated code, do not change without consulting 'Schneider Electric Automation GmbH' - otherwise you risk instability!!!*)

(* System generated code, could be modified for your application *)
Init_Exceptions();
(* End of system generated code, could be modified for your application *)

(* System generated code, do not change without consulting 'Schneider Electric Automation GmbH' - otherwise you risk instability!!!*)
Init_SubModules();
Init_CmdTables();
Init_Reactions();
UpdateStructs();
(* End of system generated code, do not change without consulting 'Schneider Electric Automation GmbH' - otherwise you risk instability!!!*)

(* System generated code, could be modified for your application *)
Init_Alpha();
Init_Bravo();
Init_Charly();
Init_NodeWithoutMotion();
(* End of system generated code, could be modified for your application *)

(* Application specific code *)
(* ToDo: Add your application specific code here *)
;
(* End of application specific code *)
END_ACTION

ACTION Input_Action:
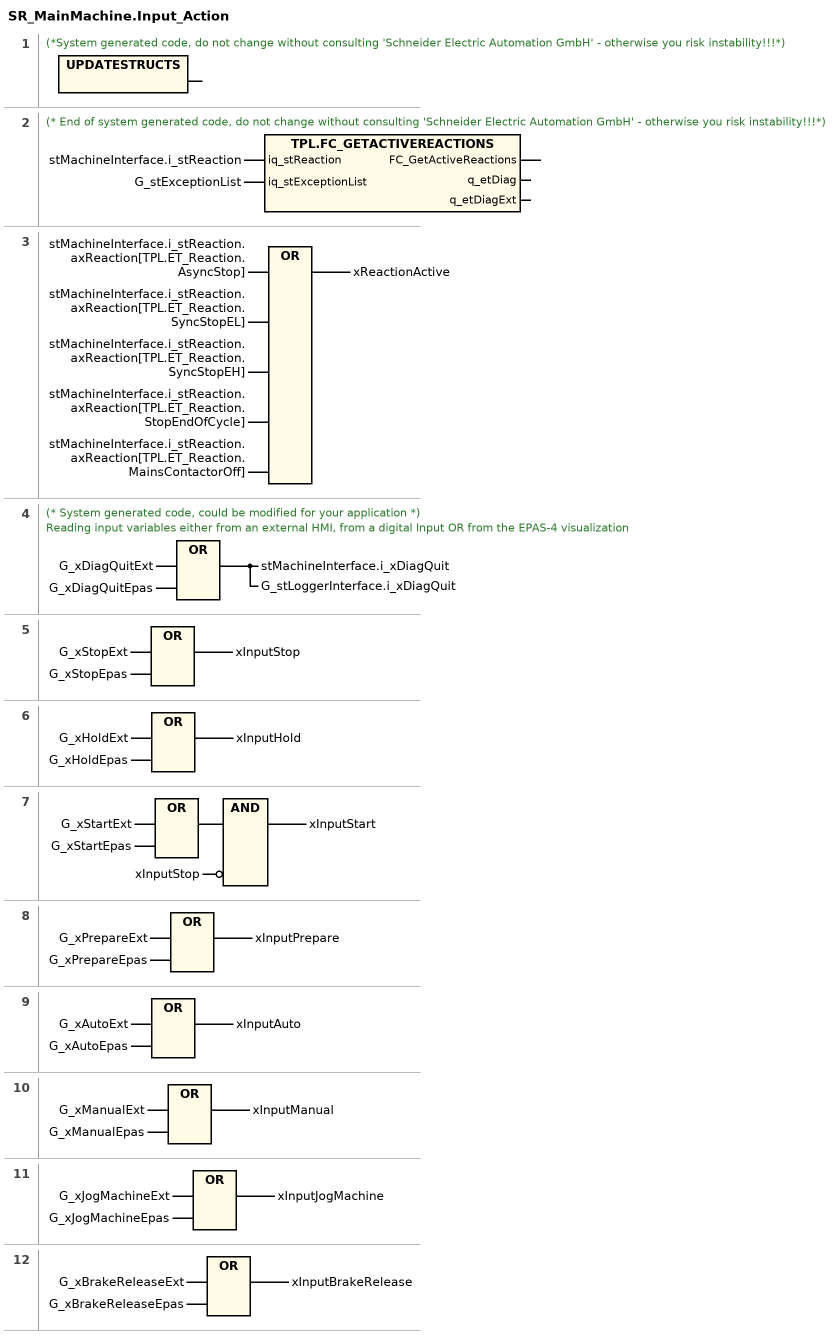
// NETWORK 1
// (*System generated code, do not change without consulting 'Schneider Electric Automation GmbH' - otherwise you risk instability!!!*)
UPDATESTRUCTS();

// NETWORK 2
// (* End of system generated code, do not change without consulting 'Schneider Electric Automation GmbH' - otherwise you risk instability!!!*)
TPL.FC_GETACTIVEREACTIONS(iq_stReaction := stMachineInterface.i_stReaction, iq_stExceptionList := G_stExceptionList);

// NETWORK 3
xReactionActive := stMachineInterface.i_stReaction.axReaction[TPL.ET_Reaction.AsyncStop] OR stMachineInterface.i_stReaction.axReaction[TPL.ET_Reaction.SyncStopEL] OR stMachineInterface.i_stReaction.axReaction[TPL.ET_Reaction.SyncStopEH] OR stMachineInterface.i_stReaction.axReaction[TPL.ET_Reaction.StopEndOfCycle] OR stMachineInterface.i_stReaction.axReaction[TPL.ET_Reaction.MainsContactorOff];

// NETWORK 4
// 					(* System generated code, could be modified for your application *)
// Reading input variables either from an external HMI, from a digital Input OR from the EPAS-4 visualization
//
_w1 := G_xDiagQuitExt OR G_xDiagQuitEpas;
stMachineInterface.i_xDiagQuit := _w1;
G_stLoggerInterface.i_xDiagQuit := _w1;

// NETWORK 5
xInputStop := G_xStopExt OR G_xStopEpas;

// NETWORK 6
xInputHold := G_xHoldExt OR G_xHoldEpas;

// NETWORK 7
xInputStart := (G_xStartExt OR G_xStartEpas) AND NOT xInputStop;

// NETWORK 8
xInputPrepare := G_xPrepareExt OR G_xPrepareEpas;

// NETWORK 9
xInputAuto := G_xAutoExt OR G_xAutoEpas;

// NETWORK 10
xInputManual := G_xManualExt OR G_xManualEpas;

// NETWORK 11
xInputJogMachine := G_xJogMachineExt OR G_xJogMachineEpas;

// NETWORK 12
xInputBrakeRelease := G_xBrakeReleaseExt OR G_xBrakeReleaseEpas;

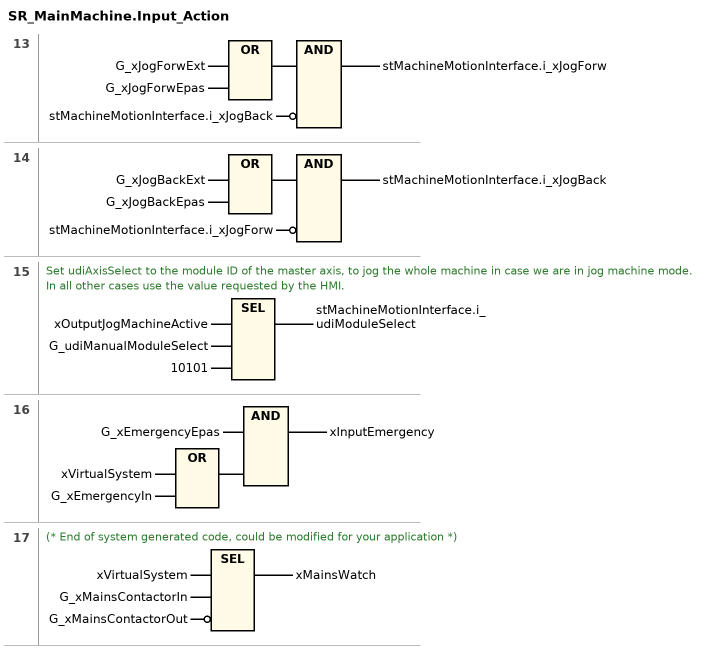
// NETWORK 13
stMachineMotionInterface.i_xJogForw := (G_xJogForwExt OR G_xJogForwEpas) AND NOT stMachineMotionInterface.i_xJogBack;

// NETWORK 14
stMachineMotionInterface.i_xJogBack := (G_xJogBackExt OR G_xJogBackEpas) AND NOT stMachineMotionInterface.i_xJogForw;

// NETWORK 15
// 					Set udiAxisSelect to the module ID of the master axis, to jog the whole machine in case we are in jog machine mode.
// In all other cases use the value requested by the HMI.
//
stMachineMotionInterface.i_udiModuleSelect := SEL(xOutputJogMachineActive, G_udiManualModuleSelect, 10101);

// NETWORK 16
xInputEmergency := G_xEmergencyEpas AND (xVirtualSystem OR G_xEmergencyIn);

// NETWORK 17
// (* End of system generated code, could be modified for your application *)
xMainsWatch := SEL(xVirtualSystem, G_xMainsContactorIn, NOT G_xMainsContactorOut);
END_ACTION

ACTION JogMachineStep_Action:
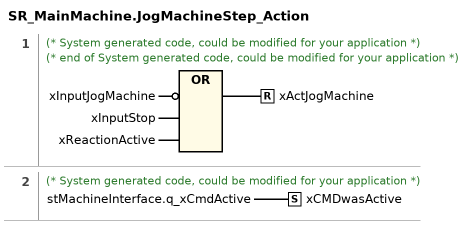
// NETWORK 1
// 					(* System generated code, could be modified for your application *)
// (* end of System generated code, could be modified for your application *)
//
xActJogMachine R= NOT xInputJogMachine OR xInputStop OR xReactionActive;

// NETWORK 2
// (* System generated code, could be modified for your application *)
xCMDwasActive S= stMachineInterface.q_xCmdActive;
END_ACTION

ACTION JogMachineStep_Entry:
(* System generated code, could be modified for your application *)
	xCMDwasActive		:=FALSE;
	stMachineInterface.iq_diCmd	:= ET_Cmd.Jogging;
(* End of system generated code, could be modified for your application *)
END_ACTION

ACTION Logger_Action:
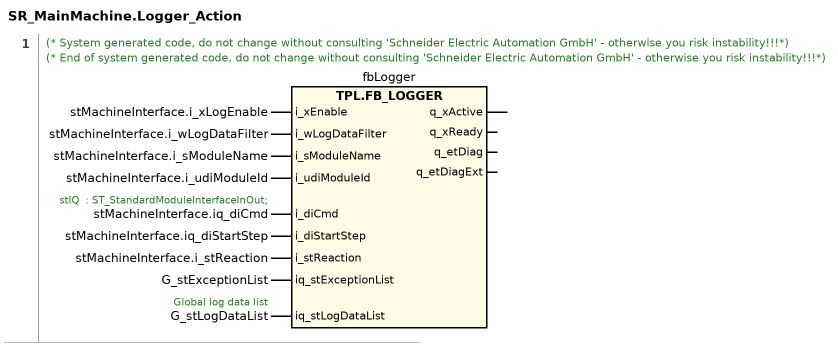
// NETWORK 1
// 					(* System generated code, do not change without consulting 'Schneider Electric Automation GmbH' - otherwise you risk instability!!!*)
// (* End of system generated code, do not change without consulting 'Schneider Electric Automation GmbH' - otherwise you risk instability!!!*)
//
//   fbLogger: Logging related variables
//   stMachineInterface.iq_diCmd: stIQ : ST_StandardModuleInterfaceInOut;
//   G_stLogDataList: Global log data list
fbLogger(
    i_xEnable := stMachineInterface.i_xLogEnable,
    i_wLogDataFilter := stMachineInterface.i_wLogDataFilter,
    i_sModuleName := stMachineInterface.i_sModuleName,
    i_udiModuleId := stMachineInterface.i_udiModuleId,
    i_diCmd := stMachineInterface.iq_diCmd,
    i_diStartStep := stMachineInterface.iq_diStartStep,
    i_stReaction := stMachineInterface.i_stReaction,
    iq_stExceptionList := G_stExceptionList,
    iq_stLogDataList := G_stLogDataList); // TPL.FB_LOGGER
END_ACTION

ACTION Logic_active:
;
END_ACTION

ACTION MainSystemFaults:
(* System generated code, do not change without consulting 'Schneider Electric Automation GmbH' - otherwise you risk instability!!! *)

fbControllerDiag.Get(	q_diObjectType		=> diObjectType,
						q_sTypeName			=> sTypeName,
						q_diObjectInstance	=> diObjectInstance,
						q_sInstanceName		=> sInstanceName,
						q_diDiagCode		=> diDiagCode,
						q_diDiagClass		=> diDiagClass,
						q_diDiagNumber		=> diDiagNum,
						q_sDiagMsg			=> sDiagMsg,
						q_xHWReset			=> xHWReset);

IF diDiagClass = 4 AND diObjectType <> 32900 THEN

	IF SYSTEMCONFIGURATION.G_ifController <> 0 THEN
		sDiagMsg := SYSTEMCONFIGURATION.G_ifController.DiagMsg;
	END_IF
	
	stSystemException1.etDiag		:= GD.ET_Diag.DiagActive;
	stSystemException1.udiDiagExt	:= ET_DiagExt.SystemFatalException;								
	stSystemException1.sDiagExt		:= FC_EtDiagExtToString(stSystemException1.udiDiagExt);	
	stSystemException1.sMsg			:= PDL.FC_MultiConcat(	i_sString1 := STANDARD.CONCAT('DiagCode ', DINT_TO_STRING(diDiagCode)),
															i_sString2 := STANDARD.CONCAT(' - DiagMsg', sDiagMsg), 
															i_sString3 :=  STANDARD.CONCAT(' - ', sInstanceName), 
															i_sString4 := '');
	TPL.FC_SetException(i_xExceptionActive	:= TRUE,
						iq_stException		:= stSystemException1,
						iq_stExceptionList	:= G_stExceptionList,
						iq_stLogDataList	:= G_stLogDataList);
	
	ELSIF diDiagClass = 3 AND diObjectType <> 32900 THEN
	
	IF SYSTEMCONFIGURATION.G_ifController <> 0 THEN
		sDiagMsg := SYSTEMCONFIGURATION.G_ifController.DiagMsg;
	END_IF
	
	stSystemException2.etDiag		:= GD.ET_Diag.DiagActive;
	stSystemException2.udiDiagExt	:= ET_DiagExt.SystemException;				
	stSystemException2.sDiagExt		:= FC_EtDiagExtToString(stSystemException2.udiDiagExt);	
	stSystemException2.sMsg			:= PDL.FC_MultiConcat(	i_sString1 := STANDARD.CONCAT('DiagCode ', DINT_TO_STRING(diDiagCode)),
															i_sString2 := STANDARD.CONCAT(' - DiagMsg', sDiagMsg), 
															i_sString3 :=  STANDARD.CONCAT(' - ',sInstanceName),
															i_sString4 := '');
	TPL.FC_SetException(i_xExceptionActive	:= TRUE,
						iq_stException		:= stSystemException2,
						iq_stExceptionList	:= G_stExceptionList,
						iq_stLogDataList	:= G_stLogDataList);
	
	ELSIF (diDiagClass = 2 OR diDiagClass = 1) AND diObjectType <> 32900 THEN
	
	IF SYSTEMCONFIGURATION.G_ifController <> 0 THEN
		sDiagMsg := SYSTEMCONFIGURATION.G_ifController.DiagMsg;
	END_IF

	stSystemException3.etDiag		:= GD.ET_Diag.DiagActive;
	stSystemException3.udiDiagExt	:= ET_DiagExt.SystemWarning;
	stSystemException3.sDiagExt		:= FC_EtDiagExtToString(stSystemException3.udiDiagExt);	
	stSystemException3.sMsg			:= PDL.FC_MultiConcat(	i_sString1 := STANDARD.CONCAT('DiagCode ', DINT_TO_STRING(diDiagCode)),
															i_sString2 := STANDARD.CONCAT(' - DiagMsg', sDiagMsg), 
															i_sString3 := STANDARD.CONCAT(' - ',sInstanceName),
															i_sString4 := '');
	TPL.FC_SetException(i_xExceptionActive	:= TRUE,
						iq_stException		:= stSystemException3,
						iq_stExceptionList	:= G_stExceptionList,
						iq_stLogDataList	:= G_stLogDataList);
END_IF

IF NOT xInputEmergency THEN	(* Extend logic for hardware *)

	TPL.FC_SetException(i_xExceptionActive	:= TRUE,
						iq_stException		:= stEmergencyStopException,
						iq_stExceptionList	:= G_stExceptionList,
						iq_stLogDataList	:= G_stLogDataList);
END_IF

IF etContactorControlDiag <> GD.ET_Diag.Ok THEN

	stContactorControlException.etDiag		:= etContactorControlDiag;
	stContactorControlException.udiDiagExt	:= etContactorControlDiagExt;
	stContactorControlException.sDiagExt	:= TPL.FC_EtDiagExtToString(etContactorControlDiagExt);
	stContactorControlException.sMsg		:= sContactorControlMsg;
	
	TPL.FC_SetException(i_xExceptionActive	:= TRUE,
						iq_stException		:= stContactorControlException,
						iq_stExceptionList	:= G_stExceptionList,
						iq_stLogDataList	:= G_stLogDataList);
END_IF

(* End of system generated code, do not change without consulting 'Schneider Electric Automation GmbH' - otherwise you risk instability!!! *)
END_ACTION

ACTION MainUserFaults:
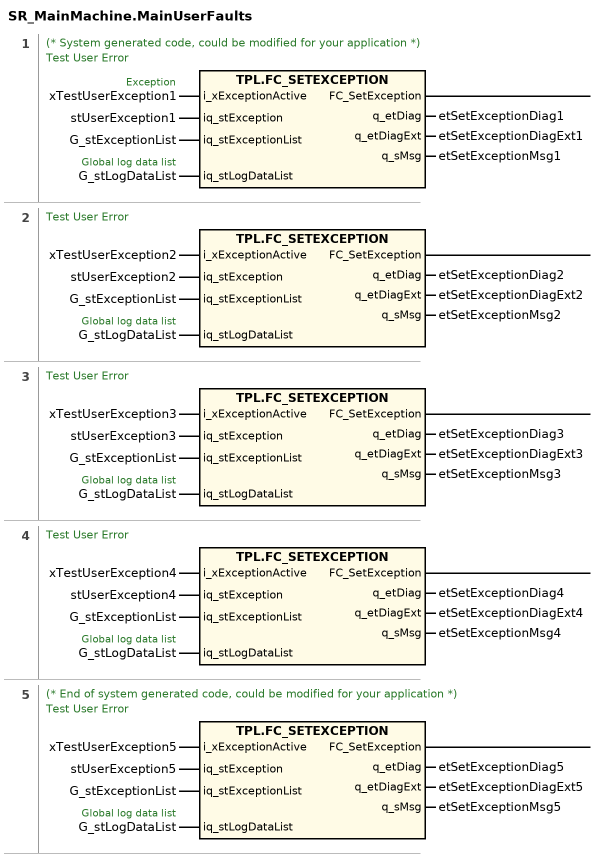
// NETWORK 1
// 					(* System generated code, could be modified for your application *)
// Test User Error
//
//   xTestUserException1: Exception
//   G_stLogDataList: Global log data list
TPL.FC_SETEXCEPTION(i_xExceptionActive := xTestUserException1, iq_stException := stUserException1, iq_stExceptionList := G_stExceptionList, iq_stLogDataList := G_stLogDataList, q_etDiag => etSetExceptionDiag1, q_etDiagExt => etSetExceptionDiagExt1, q_sMsg => etSetExceptionMsg1);

// NETWORK 2
// Test User Error
//   G_stLogDataList: Global log data list
TPL.FC_SETEXCEPTION(i_xExceptionActive := xTestUserException2, iq_stException := stUserException2, iq_stExceptionList := G_stExceptionList, iq_stLogDataList := G_stLogDataList, q_etDiag => etSetExceptionDiag2, q_etDiagExt => etSetExceptionDiagExt2, q_sMsg => etSetExceptionMsg2);

// NETWORK 3
// Test User Error
//   G_stLogDataList: Global log data list
TPL.FC_SETEXCEPTION(i_xExceptionActive := xTestUserException3, iq_stException := stUserException3, iq_stExceptionList := G_stExceptionList, iq_stLogDataList := G_stLogDataList, q_etDiag => etSetExceptionDiag3, q_etDiagExt => etSetExceptionDiagExt3, q_sMsg => etSetExceptionMsg3);

// NETWORK 4
// Test User Error
//   G_stLogDataList: Global log data list
TPL.FC_SETEXCEPTION(i_xExceptionActive := xTestUserException4, iq_stException := stUserException4, iq_stExceptionList := G_stExceptionList, iq_stLogDataList := G_stLogDataList, q_etDiag => etSetExceptionDiag4, q_etDiagExt => etSetExceptionDiagExt4, q_sMsg => etSetExceptionMsg4);

// NETWORK 5
// 					(* End of system generated code, could be modified for your application *)
// Test User Error
//
//   G_stLogDataList: Global log data list
TPL.FC_SETEXCEPTION(i_xExceptionActive := xTestUserException5, iq_stException := stUserException5, iq_stExceptionList := G_stExceptionList, iq_stLogDataList := G_stLogDataList, q_etDiag => etSetExceptionDiag5, q_etDiagExt => etSetExceptionDiagExt5, q_sMsg => etSetExceptionMsg5);
END_ACTION

ACTION ManualStep_Action:
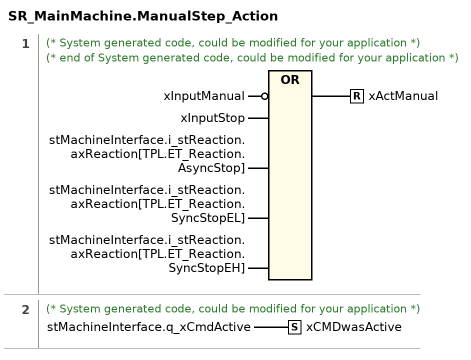
// NETWORK 1
// 					(* System generated code, could be modified for your application *)
// (* end of System generated code, could be modified for your application *)
//
xActManual R= NOT xInputManual OR xInputStop OR stMachineInterface.i_stReaction.axReaction[TPL.ET_Reaction.AsyncStop] OR stMachineInterface.i_stReaction.axReaction[TPL.ET_Reaction.SyncStopEL] OR stMachineInterface.i_stReaction.axReaction[TPL.ET_Reaction.SyncStopEH];

// NETWORK 2
// (* System generated code, could be modified for your application *)
xCMDwasActive S= stMachineInterface.q_xCmdActive;
END_ACTION

ACTION ManualStep_Entry:
(* System generated code, could be modified for your application *)
	xCMDwasActive := FALSE;
	stMachineInterface.iq_diCmd	:= ET_Cmd.Manual;
(* End of system generated code, could be modified for your application *)
END_ACTION

ACTION ModeSelect_Action:
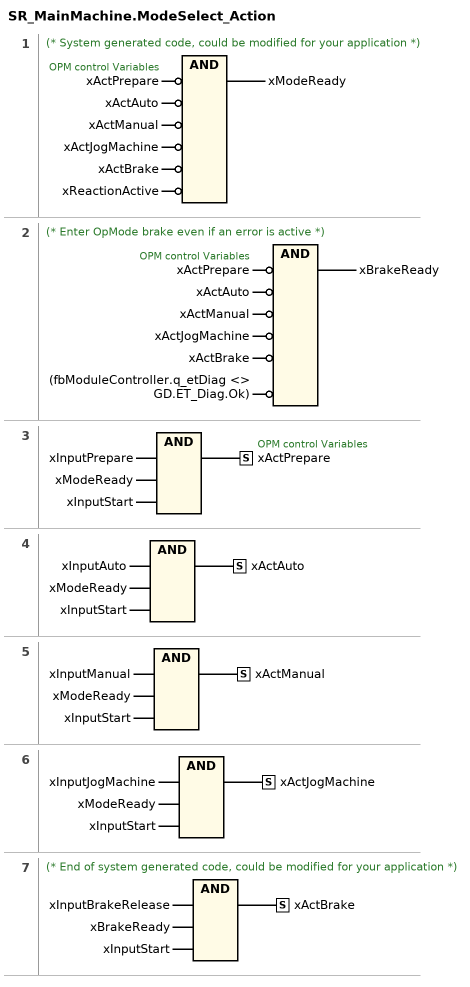
// NETWORK 1
// (* System generated code, could be modified for your application *)
//   xActPrepare: OPM control Variables
xModeReady := NOT xActPrepare AND NOT xActAuto AND NOT xActManual AND NOT xActJogMachine AND NOT xActBrake AND NOT xReactionActive;

// NETWORK 2
// (* Enter OpMode brake even if an error is active *)
//   xActPrepare: OPM control Variables
xBrakeReady := NOT xActPrepare AND NOT xActAuto AND NOT xActManual AND NOT xActJogMachine AND NOT xActBrake AND NOT ((fbModuleController.q_etDiag <> GD.ET_Diag.Ok));

// NETWORK 3
//   xActPrepare: OPM control Variables
xActPrepare S= xInputPrepare AND xModeReady AND xInputStart;

// NETWORK 4
xActAuto S= xInputAuto AND xModeReady AND xInputStart;

// NETWORK 5
xActManual S= xInputManual AND xModeReady AND xInputStart;

// NETWORK 6
xActJogMachine S= xInputJogMachine AND xModeReady AND xInputStart;

// NETWORK 7
// (* End of system generated code, could be modified for your application *)
xActBrake S= xInputBrakeRelease AND xBrakeReady AND xInputStart;
END_ACTION

ACTION Output_Action:
(* System generated code, could be modified for your application *)
xOutputPrepareActive	:= xActPrepare;
xOutputAutoActive		:= xActAuto;
xOutputManualActive		:= xActManual;
xOutputJogMachineActive	:= xActJogMachine;

IF stMachineInterface.q_udiSubModuleInException <> 0 THEN
	stMachineInterface.q_etDiag		:= GD.ET_Diag.Ok;
	stMachineInterface.q_udiDiagExt	:= ET_DiagExt.SubModuleInException;
	stMachineInterface.q_sDiagExt		:= FC_EtDiagExtToString(i_etDiagExt := ET_DiagExt.SubModuleInException);
	stMachineInterface.q_sMsg			:= '';
ELSE
	IF etDiagModuleController = GD.ET_Diag.Ok THEN
		stMachineInterface.q_etDiag	:= etDiagModuleController;
		stMachineInterface.q_sMsg		:= sMsgModuleController;
		
